   STATUS[439].EXT.AlarmSuppressed := FALSE;
   STATUS[439].EXT.AlarmPresent := FALSE;
   STATUS[439].EXT.AlarmFailUnAck := FALSE;
   STATUS[439].Status := 0;
   STATUS[439].TimeStamp := 16#0000;
   STATUS[440].EXT.AlarmWarnUnAck := FALSE;
   STATUS[440].EXT.AckRequired := FALSE;
   STATUS[440].EXT.Maintanence := FALSE;
   STATUS[440].EXT.Operation := FALSE;
   STATUS[440].EXT.Forced := FALSE;
   STATUS[440].EXT.BIT29 := FALSE;
   STATUS[440].EXT.BIT30 := FALSE;
   STATUS[440].EXT.BIT31 := FALSE;
   STATUS[440].EXT.ModeBit1 := FALSE;
   STATUS[440].EXT.ModeBit2 := FALSE;
   STATUS[440].EXT.ModeBit3 := FALSE;
   STATUS[440].EXT.BIT19 := FALSE;
   STATUS[440].EXT.BIT20 := FALSE;
   STATUS[440].EXT.AlarmSuppressed := FALSE;
   STATUS[440].EXT.AlarmPresent := FALSE;
   STATUS[440].EXT.AlarmFailUnAck := FALSE;
   STATUS[440].Status := 0;
   STATUS[440].TimeStamp := 16#0000;
   STATUS[441].EXT.AlarmWarnUnAck := FALSE;
   STATUS[441].EXT.AckRequired := FALSE;
   STATUS[441].EXT.Maintanence := FALSE;
   STATUS[441].EXT.Operation := FALSE;
   STATUS[441].EXT.Forced := FALSE;
   STATUS[441].EXT.BIT29 := FALSE;
   STATUS[441].EXT.BIT30 := FALSE;
   STATUS[441].EXT.BIT31 := FALSE;
   STATUS[441].EXT.ModeBit1 := FALSE;
   STATUS[441].EXT.ModeBit2 := FALSE;
   STATUS[441].EXT.ModeBit3 := FALSE;
   STATUS[441].EXT.BIT19 := FALSE;
   STATUS[441].EXT.BIT20 := FALSE;
   STATUS[441].EXT.AlarmSuppressed := FALSE;
   STATUS[441].EXT.AlarmPresent := FALSE;
   STATUS[441].EXT.AlarmFailUnAck := FALSE;
   STATUS[441].Status := 0;
   STATUS[441].TimeStamp := 16#0000;
   STATUS[442].EXT.AlarmWarnUnAck := FALSE;
   STATUS[442].EXT.AckRequired := FALSE;
   STATUS[442].EXT.Maintanence := FALSE;
   STATUS[442].EXT.Operation := FALSE;
   STATUS[442].EXT.Forced := FALSE;
   STATUS[442].EXT.BIT29 := FALSE;
   STATUS[442].EXT.BIT30 := FALSE;
   STATUS[442].EXT.BIT31 := FALSE;
   STATUS[442].EXT.ModeBit1 := FALSE;
   STATUS[442].EXT.ModeBit2 := FALSE;
   STATUS[442].EXT.ModeBit3 := FALSE;
   STATUS[442].EXT.BIT19 := FALSE;
   STATUS[442].EXT.BIT20 := FALSE;
   STATUS[442].EXT.AlarmSuppressed := FALSE;
   STATUS[442].EXT.AlarmPresent := FALSE;
   STATUS[442].EXT.AlarmFailUnAck := FALSE;
   STATUS[442].Status := 0;
   STATUS[442].TimeStamp := 16#0000;
   STATUS[443].EXT.AlarmWarnUnAck := FALSE;
   STATUS[443].EXT.AckRequired := FALSE;
   STATUS[443].EXT.Maintanence := FALSE;
   STATUS[443].EXT.Operation := FALSE;
   STATUS[443].EXT.Forced := FALSE;
   STATUS[443].EXT.BIT29 := FALSE;
   STATUS[443].EXT.BIT30 := FALSE;
   STATUS[443].EXT.BIT31 := FALSE;
   STATUS[443].EXT.ModeBit1 := FALSE;
   STATUS[443].EXT.ModeBit2 := FALSE;
   STATUS[443].EXT.ModeBit3 := FALSE;
   STATUS[443].EXT.BIT19 := FALSE;
   STATUS[443].EXT.BIT20 := FALSE;
   STATUS[443].EXT.AlarmSuppressed := FALSE;
   STATUS[443].EXT.AlarmPresent := FALSE;
   STATUS[443].EXT.AlarmFailUnAck := FALSE;
   STATUS[443].Status := 0;
   STATUS[443].TimeStamp := 16#0000;
   STATUS[444].EXT.AlarmWarnUnAck := FALSE;
   STATUS[444].EXT.AckRequired := FALSE;
   STATUS[444].EXT.Maintanence := FALSE;
   STATUS[444].EXT.Operation := FALSE;
   STATUS[444].EXT.Forced := FALSE;
   STATUS[444].EXT.BIT29 := FALSE;
   STATUS[444].EXT.BIT30 := FALSE;
   STATUS[444].EXT.BIT31 := FALSE;
   STATUS[444].EXT.ModeBit1 := FALSE;
   STATUS[444].EXT.ModeBit2 := FALSE;
   STATUS[444].EXT.ModeBit3 := FALSE;
   STATUS[444].EXT.BIT19 := FALSE;
   STATUS[444].EXT.BIT20 := FALSE;
   STATUS[444].EXT.AlarmSuppressed := FALSE;
   STATUS[444].EXT.AlarmPresent := FALSE;
   STATUS[444].EXT.AlarmFailUnAck := FALSE;
   STATUS[444].Status := 0;
   STATUS[444].TimeStamp := 16#0000;
   STATUS[445].EXT.AlarmWarnUnAck := FALSE;
   STATUS[445].EXT.AckRequired := FALSE;
   STATUS[445].EXT.Maintanence := FALSE;
   STATUS[445].EXT.Operation := FALSE;
   STATUS[445].EXT.Forced := FALSE;
   STATUS[445].EXT.BIT29 := FALSE;
   STATUS[445].EXT.BIT30 := FALSE;
   STATUS[445].EXT.BIT31 := FALSE;
   STATUS[445].EXT.ModeBit1 := FALSE;
   STATUS[445].EXT.ModeBit2 := FALSE;
   STATUS[445].EXT.ModeBit3 := FALSE;
   STATUS[445].EXT.BIT19 := FALSE;
   STATUS[445].EXT.BIT20 := FALSE;
   STATUS[445].EXT.AlarmSuppressed := FALSE;
   STATUS[445].EXT.AlarmPresent := FALSE;
   STATUS[445].EXT.AlarmFailUnAck := FALSE;
   STATUS[445].Status := 0;
   STATUS[445].TimeStamp := 16#0000;
   STATUS[446].EXT.AlarmWarnUnAck := FALSE;
   STATUS[446].EXT.AckRequired := FALSE;
   STATUS[446].EXT.Maintanence := FALSE;
   STATUS[446].EXT.Operation := FALSE;
   STATUS[446].EXT.Forced := FALSE;
   STATUS[446].EXT.BIT29 := FALSE;
   STATUS[446].EXT.BIT30 := FALSE;
   STATUS[446].EXT.BIT31 := FALSE;
   STATUS[446].EXT.ModeBit1 := FALSE;
   STATUS[446].EXT.ModeBit2 := FALSE;
   STATUS[446].EXT.ModeBit3 := FALSE;
   STATUS[446].EXT.BIT19 := FALSE;
   STATUS[446].EXT.BIT20 := FALSE;
   STATUS[446].EXT.AlarmSuppressed := FALSE;
   STATUS[446].EXT.AlarmPresent := FALSE;
   STATUS[446].EXT.AlarmFailUnAck := FALSE;
   STATUS[446].Status := 0;
   STATUS[446].TimeStamp := 16#0000;
   STATUS[447].EXT.AlarmWarnUnAck := FALSE;
   STATUS[447].EXT.AckRequired := FALSE;
   STATUS[447].EXT.Maintanence := FALSE;
   STATUS[447].EXT.Operation := FALSE;
   STATUS[447].EXT.Forced := FALSE;
   STATUS[447].EXT.BIT29 := FALSE;
   STATUS[447].EXT.BIT30 := FALSE;
   STATUS[447].EXT.BIT31 := FALSE;
   STATUS[447].EXT.ModeBit1 := FALSE;
   STATUS[447].EXT.ModeBit2 := FALSE;
   STATUS[447].EXT.ModeBit3 := FALSE;
   STATUS[447].EXT.BIT19 := FALSE;
   STATUS[447].EXT.BIT20 := FALSE;
   STATUS[447].EXT.AlarmSuppressed := FALSE;
   STATUS[447].EXT.AlarmPresent := FALSE;
   STATUS[447].EXT.AlarmFailUnAck := FALSE;
   STATUS[447].Status := 0;
   STATUS[447].TimeStamp := 16#0000;
   STATUS[448].EXT.AlarmWarnUnAck := FALSE;
   STATUS[448].EXT.AckRequired := FALSE;
   STATUS[448].EXT.Maintanence := FALSE;
   STATUS[448].EXT.Operation := FALSE;
   STATUS[448].EXT.Forced := FALSE;
   STATUS[448].EXT.BIT29 := FALSE;
   STATUS[448].EXT.BIT30 := FALSE;
   STATUS[448].EXT.BIT31 := FALSE;
   STATUS[448].EXT.ModeBit1 := FALSE;
   STATUS[448].EXT.ModeBit2 := FALSE;
   STATUS[448].EXT.ModeBit3 := FALSE;
   STATUS[448].EXT.BIT19 := FALSE;
   STATUS[448].EXT.BIT20 := FALSE;
   STATUS[448].EXT.AlarmSuppressed := FALSE;
   STATUS[448].EXT.AlarmPresent := FALSE;
   STATUS[448].EXT.AlarmFailUnAck := FALSE;
   STATUS[448].Status := 0;
   STATUS[448].TimeStamp := 16#0000;
   STATUS[449].EXT.AlarmWarnUnAck := FALSE;
   STATUS[449].EXT.AckRequired := FALSE;
   STATUS[449].EXT.Maintanence := FALSE;
   STATUS[449].EXT.Operation := FALSE;
   STATUS[449].EXT.Forced := FALSE;
   STATUS[449].EXT.BIT29 := FALSE;
   STATUS[449].EXT.BIT30 := FALSE;
   STATUS[449].EXT.BIT31 := FALSE;
   STATUS[449].EXT.ModeBit1 := FALSE;
   STATUS[449].EXT.ModeBit2 := FALSE;
   STATUS[449].EXT.ModeBit3 := FALSE;
   STATUS[449].EXT.BIT19 := FALSE;
   STATUS[449].EXT.BIT20 := FALSE;
   STATUS[449].EXT.AlarmSuppressed := FALSE;
   STATUS[449].EXT.AlarmPresent := FALSE;
   STATUS[449].EXT.AlarmFailUnAck := FALSE;
   STATUS[449].Status := 0;
   STATUS[449].TimeStamp := 16#0000;
   STATUS[450].EXT.AlarmWarnUnAck := FALSE;
   STATUS[450].EXT.AckRequired := FALSE;
   STATUS[450].EXT.Maintanence := FALSE;
   STATUS[450].EXT.Operation := FALSE;
   STATUS[450].EXT.Forced := FALSE;
   STATUS[450].EXT.BIT29 := FALSE;
   STATUS[450].EXT.BIT30 := FALSE;
   STATUS[450].EXT.BIT31 := FALSE;
   STATUS[450].EXT.ModeBit1 := FALSE;
   STATUS[450].EXT.ModeBit2 := FALSE;
   STATUS[450].EXT.ModeBit3 := FALSE;
   STATUS[450].EXT.BIT19 := FALSE;
   STATUS[450].EXT.BIT20 := FALSE;
   STATUS[450].EXT.AlarmSuppressed := FALSE;
   STATUS[450].EXT.AlarmPresent := FALSE;
   STATUS[450].EXT.AlarmFailUnAck := FALSE;
   STATUS[450].Status := 0;
   STATUS[450].TimeStamp := 16#0000;
   STATUS[451].EXT.AlarmWarnUnAck := FALSE;
   STATUS[451].EXT.AckRequired := FALSE;
   STATUS[451].EXT.Maintanence := FALSE;
   STATUS[451].EXT.Operation := FALSE;
   STATUS[451].EXT.Forced := FALSE;
   STATUS[451].EXT.BIT29 := FALSE;
   STATUS[451].EXT.BIT30 := FALSE;
   STATUS[451].EXT.BIT31 := FALSE;
   STATUS[451].EXT.ModeBit1 := FALSE;
   STATUS[451].EXT.ModeBit2 := FALSE;
   STATUS[451].EXT.ModeBit3 := FALSE;
   STATUS[451].EXT.BIT19 := FALSE;
   STATUS[451].EXT.BIT20 := FALSE;
   STATUS[451].EXT.AlarmSuppressed := FALSE;
   STATUS[451].EXT.AlarmPresent := FALSE;
   STATUS[451].EXT.AlarmFailUnAck := FALSE;
   STATUS[451].Status := 0;
   STATUS[451].TimeStamp := 16#0000;
   STATUS[452].EXT.AlarmWarnUnAck := FALSE;
   STATUS[452].EXT.AckRequired := FALSE;
   STATUS[452].EXT.Maintanence := FALSE;
   STATUS[452].EXT.Operation := FALSE;
   STATUS[452].EXT.Forced := FALSE;
   STATUS[452].EXT.BIT29 := FALSE;
   STATUS[452].EXT.BIT30 := FALSE;
   STATUS[452].EXT.BIT31 := FALSE;
   STATUS[452].EXT.ModeBit1 := FALSE;
   STATUS[452].EXT.ModeBit2 := FALSE;
   STATUS[452].EXT.ModeBit3 := FALSE;
   STATUS[452].EXT.BIT19 := FALSE;
   STATUS[452].EXT.BIT20 := FALSE;
   STATUS[452].EXT.AlarmSuppressed := FALSE;
   STATUS[452].EXT.AlarmPresent := FALSE;
   STATUS[452].EXT.AlarmFailUnAck := FALSE;
   STATUS[452].Status := 0;
   STATUS[452].TimeStamp := 16#0000;
   STATUS[453].EXT.AlarmWarnUnAck := FALSE;
   STATUS[453].EXT.AckRequired := FALSE;
   STATUS[453].EXT.Maintanence := FALSE;
   STATUS[453].EXT.Operation := FALSE;
   STATUS[453].EXT.Forced := FALSE;
   STATUS[453].EXT.BIT29 := FALSE;
   STATUS[453].EXT.BIT30 := FALSE;
   STATUS[453].EXT.BIT31 := FALSE;
   STATUS[453].EXT.ModeBit1 := FALSE;
   STATUS[453].EXT.ModeBit2 := FALSE;
   STATUS[453].EXT.ModeBit3 := FALSE;
   STATUS[453].EXT.BIT19 := FALSE;
   STATUS[453].EXT.BIT20 := FALSE;
   STATUS[453].EXT.AlarmSuppressed := FALSE;
   STATUS[453].EXT.AlarmPresent := FALSE;
   STATUS[453].EXT.AlarmFailUnAck := FALSE;
   STATUS[453].Status := 0;
   STATUS[453].TimeStamp := 16#0000;
   STATUS[454].EXT.AlarmWarnUnAck := FALSE;
   STATUS[454].EXT.AckRequired := FALSE;
   STATUS[454].EXT.Maintanence := FALSE;
   STATUS[454].EXT.Operation := FALSE;
   STATUS[454].EXT.Forced := FALSE;
   STATUS[454].EXT.BIT29 := FALSE;
   STATUS[454].EXT.BIT30 := FALSE;
   STATUS[454].EXT.BIT31 := FALSE;
   STATUS[454].EXT.ModeBit1 := FALSE;
   STATUS[454].EXT.ModeBit2 := FALSE;
   STATUS[454].EXT.ModeBit3 := FALSE;
   STATUS[454].EXT.BIT19 := FALSE;
   STATUS[454].EXT.BIT20 := FALSE;
   STATUS[454].EXT.AlarmSuppressed := FALSE;
   STATUS[454].EXT.AlarmPresent := FALSE;
   STATUS[454].EXT.AlarmFailUnAck := FALSE;
   STATUS[454].Status := 0;
   STATUS[454].TimeStamp := 16#0000;
   STATUS[455].EXT.AlarmWarnUnAck := FALSE;
   STATUS[455].EXT.AckRequired := FALSE;
   STATUS[455].EXT.Maintanence := FALSE;
   STATUS[455].EXT.Operation := FALSE;
   STATUS[455].EXT.Forced := FALSE;
   STATUS[455].EXT.BIT29 := FALSE;
   STATUS[455].EXT.BIT30 := FALSE;
   STATUS[455].EXT.BIT31 := FALSE;
   STATUS[455].EXT.ModeBit1 := FALSE;
   STATUS[455].EXT.ModeBit2 := FALSE;
   STATUS[455].EXT.ModeBit3 := FALSE;
   STATUS[455].EXT.BIT19 := FALSE;
   STATUS[455].EXT.BIT20 := FALSE;
   STATUS[455].EXT.AlarmSuppressed := FALSE;
   STATUS[455].EXT.AlarmPresent := FALSE;
   STATUS[455].EXT.AlarmFailUnAck := FALSE;
   STATUS[455].Status := 0;
   STATUS[455].TimeStamp := 16#0000;
   STATUS[456].EXT.AlarmWarnUnAck := FALSE;
   STATUS[456].EXT.AckRequired := FALSE;
   STATUS[456].EXT.Maintanence := FALSE;
   STATUS[456].EXT.Operation := FALSE;
   STATUS[456].EXT.Forced := FALSE;
   STATUS[456].EXT.BIT29 := FALSE;
   STATUS[456].EXT.BIT30 := FALSE;
   STATUS[456].EXT.BIT31 := FALSE;
   STATUS[456].EXT.ModeBit1 := FALSE;
   STATUS[456].EXT.ModeBit2 := FALSE;
   STATUS[456].EXT.ModeBit3 := FALSE;
   STATUS[456].EXT.BIT19 := FALSE;
   STATUS[456].EXT.BIT20 := FALSE;
   STATUS[456].EXT.AlarmSuppressed := FALSE;
   STATUS[456].EXT.AlarmPresent := FALSE;
   STATUS[456].EXT.AlarmFailUnAck := FALSE;
   STATUS[456].Status := 0;
   STATUS[456].TimeStamp := 16#0000;
   STATUS[457].EXT.AlarmWarnUnAck := FALSE;
   STATUS[457].EXT.AckRequired := FALSE;
   STATUS[457].EXT.Maintanence := FALSE;
   STATUS[457].EXT.Operation := FALSE;
   STATUS[457].EXT.Forced := FALSE;
   STATUS[457].EXT.BIT29 := FALSE;
   STATUS[457].EXT.BIT30 := FALSE;
   STATUS[457].EXT.BIT31 := FALSE;
   STATUS[457].EXT.ModeBit1 := FALSE;
   STATUS[457].EXT.ModeBit2 := FALSE;
   STATUS[457].EXT.ModeBit3 := FALSE;
   STATUS[457].EXT.BIT19 := FALSE;
   STATUS[457].EXT.BIT20 := FALSE;
   STATUS[457].EXT.AlarmSuppressed := FALSE;
   STATUS[457].EXT.AlarmPresent := FALSE;
   STATUS[457].EXT.AlarmFailUnAck := FALSE;
   STATUS[457].Status := 0;
   STATUS[457].TimeStamp := 16#0000;
   STATUS[458].EXT.AlarmWarnUnAck := FALSE;
   STATUS[458].EXT.AckRequired := FALSE;
   STATUS[458].EXT.Maintanence := FALSE;
   STATUS[458].EXT.Operation := FALSE;
   STATUS[458].EXT.Forced := FALSE;
   STATUS[458].EXT.BIT29 := FALSE;
   STATUS[458].EXT.BIT30 := FALSE;
   STATUS[458].EXT.BIT31 := FALSE;
   STATUS[458].EXT.ModeBit1 := FALSE;
   STATUS[458].EXT.ModeBit2 := FALSE;
   STATUS[458].EXT.ModeBit3 := FALSE;
   STATUS[458].EXT.BIT19 := FALSE;
   STATUS[458].EXT.BIT20 := FALSE;
   STATUS[458].EXT.AlarmSuppressed := FALSE;
   STATUS[458].EXT.AlarmPresent := FALSE;
   STATUS[458].EXT.AlarmFailUnAck := FALSE;
   STATUS[458].Status := 0;
   STATUS[458].TimeStamp := 16#0000;
   STATUS[459].EXT.AlarmWarnUnAck := FALSE;
   STATUS[459].EXT.AckRequired := FALSE;
   STATUS[459].EXT.Maintanence := FALSE;
   STATUS[459].EXT.Operation := FALSE;
   STATUS[459].EXT.Forced := FALSE;
   STATUS[459].EXT.BIT29 := FALSE;
   STATUS[459].EXT.BIT30 := FALSE;
   STATUS[459].EXT.BIT31 := FALSE;
   STATUS[459].EXT.ModeBit1 := FALSE;
   STATUS[459].EXT.ModeBit2 := FALSE;
   STATUS[459].EXT.ModeBit3 := FALSE;
   STATUS[459].EXT.BIT19 := FALSE;
   STATUS[459].EXT.BIT20 := FALSE;
   STATUS[459].EXT.AlarmSuppressed := FALSE;
   STATUS[459].EXT.AlarmPresent := FALSE;
   STATUS[459].EXT.AlarmFailUnAck := FALSE;
   STATUS[459].Status := 0;
   STATUS[459].TimeStamp := 16#0000;
   STATUS[460].EXT.AlarmWarnUnAck := FALSE;
   STATUS[460].EXT.AckRequired := FALSE;
   STATUS[460].EXT.Maintanence := FALSE;
   STATUS[460].EXT.Operation := FALSE;
   STATUS[460].EXT.Forced := FALSE;
   STATUS[460].EXT.BIT29 := FALSE;
   STATUS[460].EXT.BIT30 := FALSE;
   STATUS[460].EXT.BIT31 := FALSE;
   STATUS[460].EXT.ModeBit1 := FALSE;
   STATUS[460].EXT.ModeBit2 := FALSE;
   STATUS[460].EXT.ModeBit3 := FALSE;
   STATUS[460].EXT.BIT19 := FALSE;
   STATUS[460].EXT.BIT20 := FALSE;
   STATUS[460].EXT.AlarmSuppressed := FALSE;
   STATUS[460].EXT.AlarmPresent := FALSE;
   STATUS[460].EXT.AlarmFailUnAck := FALSE;
   STATUS[460].Status := 0;
   STATUS[460].TimeStamp := 16#0000;
   STATUS[461].EXT.AlarmWarnUnAck := FALSE;
   STATUS[461].EXT.AckRequired := FALSE;
   STATUS[461].EXT.Maintanence := FALSE;
   STATUS[461].EXT.Operation := FALSE;
   STATUS[461].EXT.Forced := FALSE;
   STATUS[461].EXT.BIT29 := FALSE;
   STATUS[461].EXT.BIT30 := FALSE;
   STATUS[461].EXT.BIT31 := FALSE;
   STATUS[461].EXT.ModeBit1 := FALSE;
   STATUS[461].EXT.ModeBit2 := FALSE;
   STATUS[461].EXT.ModeBit3 := FALSE;
   STATUS[461].EXT.BIT19 := FALSE;
   STATUS[461].EXT.BIT20 := FALSE;
   STATUS[461].EXT.AlarmSuppressed := FALSE;
   STATUS[461].EXT.AlarmPresent := FALSE;
   STATUS[461].EXT.AlarmFailUnAck := FALSE;
   STATUS[461].Status := 0;
   STATUS[461].TimeStamp := 16#0000;
   STATUS[462].EXT.AlarmWarnUnAck := FALSE;
   STATUS[462].EXT.AckRequired := FALSE;
   STATUS[462].EXT.Maintanence := FALSE;
   STATUS[462].EXT.Operation := FALSE;
   STATUS[462].EXT.Forced := FALSE;
   STATUS[462].EXT.BIT29 := FALSE;
   STATUS[462].EXT.BIT30 := FALSE;
   STATUS[462].EXT.BIT31 := FALSE;
   STATUS[462].EXT.ModeBit1 := FALSE;
   STATUS[462].EXT.ModeBit2 := FALSE;
   STATUS[462].EXT.ModeBit3 := FALSE;
   STATUS[462].EXT.BIT19 := FALSE;
   STATUS[462].EXT.BIT20 := FALSE;
   STATUS[462].EXT.AlarmSuppressed := FALSE;
   STATUS[462].EXT.AlarmPresent := FALSE;
   STATUS[462].EXT.AlarmFailUnAck := FALSE;
   STATUS[462].Status := 0;
   STATUS[462].TimeStamp := 16#0000;
   STATUS[463].EXT.AlarmWarnUnAck := FALSE;
   STATUS[463].EXT.AckRequired := FALSE;
   STATUS[463].EXT.Maintanence := FALSE;
   STATUS[463].EXT.Operation := FALSE;
   STATUS[463].EXT.Forced := FALSE;
   STATUS[463].EXT.BIT29 := FALSE;
   STATUS[463].EXT.BIT30 := FALSE;
   STATUS[463].EXT.BIT31 := FALSE;
   STATUS[463].EXT.ModeBit1 := FALSE;
   STATUS[463].EXT.ModeBit2 := FALSE;
   STATUS[463].EXT.ModeBit3 := FALSE;
   STATUS[463].EXT.BIT19 := FALSE;
   STATUS[463].EXT.BIT20 := FALSE;
   STATUS[463].EXT.AlarmSuppressed := FALSE;
   STATUS[463].EXT.AlarmPresent := FALSE;
   STATUS[463].EXT.AlarmFailUnAck := FALSE;
   STATUS[463].Status := 0;
   STATUS[463].TimeStamp := 16#0000;
   STATUS[464].EXT.AlarmWarnUnAck := FALSE;
   STATUS[464].EXT.AckRequired := FALSE;
   STATUS[464].EXT.Maintanence := FALSE;
   STATUS[464].EXT.Operation := FALSE;
   STATUS[464].EXT.Forced := FALSE;
   STATUS[464].EXT.BIT29 := FALSE;
   STATUS[464].EXT.BIT30 := FALSE;
   STATUS[464].EXT.BIT31 := FALSE;
   STATUS[464].EXT.ModeBit1 := FALSE;
   STATUS[464].EXT.ModeBit2 := FALSE;
   STATUS[464].EXT.ModeBit3 := FALSE;
   STATUS[464].EXT.BIT19 := FALSE;
   STATUS[464].EXT.BIT20 := FALSE;
   STATUS[464].EXT.AlarmSuppressed := FALSE;
   STATUS[464].EXT.AlarmPresent := FALSE;
   STATUS[464].EXT.AlarmFailUnAck := FALSE;
   STATUS[464].Status := 0;
   STATUS[464].TimeStamp := 16#0000;
   STATUS[465].EXT.AlarmWarnUnAck := FALSE;
   STATUS[465].EXT.AckRequired := FALSE;
   STATUS[465].EXT.Maintanence := FALSE;
   STATUS[465].EXT.Operation := FALSE;
   STATUS[465].EXT.Forced := FALSE;
   STATUS[465].EXT.BIT29 := FALSE;
   STATUS[465].EXT.BIT30 := FALSE;
   STATUS[465].EXT.BIT31 := FALSE;
   STATUS[465].EXT.ModeBit1 := FALSE;
   STATUS[465].EXT.ModeBit2 := FALSE;
   STATUS[465].EXT.ModeBit3 := FALSE;
   STATUS[465].EXT.BIT19 := FALSE;
   STATUS[465].EXT.BIT20 := FALSE;
   STATUS[465].EXT.AlarmSuppressed := FALSE;
   STATUS[465].EXT.AlarmPresent := FALSE;
   STATUS[465].EXT.AlarmFailUnAck := FALSE;
   STATUS[465].Status := 0;
   STATUS[465].TimeStamp := 16#0000;
   STATUS[466].EXT.AlarmWarnUnAck := FALSE;
   STATUS[466].EXT.AckRequired := FALSE;
   STATUS[466].EXT.Maintanence := FALSE;
   STATUS[466].EXT.Operation := FALSE;
   STATUS[466].EXT.Forced := FALSE;
   STATUS[466].EXT.BIT29 := FALSE;
   STATUS[466].EXT.BIT30 := FALSE;
   STATUS[466].EXT.BIT31 := FALSE;
   STATUS[466].EXT.ModeBit1 := FALSE;
   STATUS[466].EXT.ModeBit2 := FALSE;
   STATUS[466].EXT.ModeBit3 := FALSE;
   STATUS[466].EXT.BIT19 := FALSE;
   STATUS[466].EXT.BIT20 := FALSE;
   STATUS[466].EXT.AlarmSuppressed := FALSE;
   STATUS[466].EXT.AlarmPresent := FALSE;
   STATUS[466].EXT.AlarmFailUnAck := FALSE;
   STATUS[466].Status := 0;
   STATUS[466].TimeStamp := 16#0000;
   STATUS[467].EXT.AlarmWarnUnAck := FALSE;
   STATUS[467].EXT.AckRequired := FALSE;
   STATUS[467].EXT.Maintanence := FALSE;
   STATUS[467].EXT.Operation := FALSE;
   STATUS[467].EXT.Forced := FALSE;
   STATUS[467].EXT.BIT29 := FALSE;
   STATUS[467].EXT.BIT30 := FALSE;
   STATUS[467].EXT.BIT31 := FALSE;
   STATUS[467].EXT.ModeBit1 := FALSE;
   STATUS[467].EXT.ModeBit2 := FALSE;
   STATUS[467].EXT.ModeBit3 := FALSE;
   STATUS[467].EXT.BIT19 := FALSE;
   STATUS[467].EXT.BIT20 := FALSE;
   STATUS[467].EXT.AlarmSuppressed := FALSE;
   STATUS[467].EXT.AlarmPresent := FALSE;
   STATUS[467].EXT.AlarmFailUnAck := FALSE;
   STATUS[467].Status := 0;
   STATUS[467].TimeStamp := 16#0000;
   STATUS[468].EXT.AlarmWarnUnAck := FALSE;
   STATUS[468].EXT.AckRequired := FALSE;
   STATUS[468].EXT.Maintanence := FALSE;
   STATUS[468].EXT.Operation := FALSE;
   STATUS[468].EXT.Forced := FALSE;
   STATUS[468].EXT.BIT29 := FALSE;
   STATUS[468].EXT.BIT30 := FALSE;
   STATUS[468].EXT.BIT31 := FALSE;
   STATUS[468].EXT.ModeBit1 := FALSE;
   STATUS[468].EXT.ModeBit2 := FALSE;
   STATUS[468].EXT.ModeBit3 := FALSE;
   STATUS[468].EXT.BIT19 := FALSE;
   STATUS[468].EXT.BIT20 := FALSE;
   STATUS[468].EXT.AlarmSuppressed := FALSE;
   STATUS[468].EXT.AlarmPresent := FALSE;
   STATUS[468].EXT.AlarmFailUnAck := FALSE;
   STATUS[468].Status := 0;
   STATUS[468].TimeStamp := 16#0000;
   STATUS[469].EXT.AlarmWarnUnAck := FALSE;
   STATUS[469].EXT.AckRequired := FALSE;
   STATUS[469].EXT.Maintanence := FALSE;
   STATUS[469].EXT.Operation := FALSE;
   STATUS[469].EXT.Forced := FALSE;
   STATUS[469].EXT.BIT29 := FALSE;
   STATUS[469].EXT.BIT30 := FALSE;
   STATUS[469].EXT.BIT31 := FALSE;
   STATUS[469].EXT.ModeBit1 := FALSE;
   STATUS[469].EXT.ModeBit2 := FALSE;
   STATUS[469].EXT.ModeBit3 := FALSE;
   STATUS[469].EXT.BIT19 := FALSE;
   STATUS[469].EXT.BIT20 := FALSE;
   STATUS[469].EXT.AlarmSuppressed := FALSE;
   STATUS[469].EXT.AlarmPresent := FALSE;
   STATUS[469].EXT.AlarmFailUnAck := FALSE;
   STATUS[469].Status := 0;
   STATUS[469].TimeStamp := 16#0000;
   STATUS[470].EXT.AlarmWarnUnAck := FALSE;
   STATUS[470].EXT.AckRequired := FALSE;
   STATUS[470].EXT.Maintanence := FALSE;
   STATUS[470].EXT.Operation := FALSE;
   STATUS[470].EXT.Forced := FALSE;
   STATUS[470].EXT.BIT29 := FALSE;
   STATUS[470].EXT.BIT30 := FALSE;
   STATUS[470].EXT.BIT31 := FALSE;
   STATUS[470].EXT.ModeBit1 := FALSE;
   STATUS[470].EXT.ModeBit2 := FALSE;
   STATUS[470].EXT.ModeBit3 := FALSE;
   STATUS[470].EXT.BIT19 := FALSE;
   STATUS[470].EXT.BIT20 := FALSE;
   STATUS[470].EXT.AlarmSuppressed := FALSE;
   STATUS[470].EXT.AlarmPresent := FALSE;
   STATUS[470].EXT.AlarmFailUnAck := FALSE;
   STATUS[470].Status := 0;
   STATUS[470].TimeStamp := 16#0000;
   STATUS[471].EXT.AlarmWarnUnAck := FALSE;
   STATUS[471].EXT.AckRequired := FALSE;
   STATUS[471].EXT.Maintanence := FALSE;
   STATUS[471].EXT.Operation := FALSE;
   STATUS[471].EXT.Forced := FALSE;
   STATUS[471].EXT.BIT29 := FALSE;
   STATUS[471].EXT.BIT30 := FALSE;
   STATUS[471].EXT.BIT31 := FALSE;
   STATUS[471].EXT.ModeBit1 := FALSE;
   STATUS[471].EXT.ModeBit2 := FALSE;
   STATUS[471].EXT.ModeBit3 := FALSE;
   STATUS[471].EXT.BIT19 := FALSE;
   STATUS[471].EXT.BIT20 := FALSE;
   STATUS[471].EXT.AlarmSuppressed := FALSE;
   STATUS[471].EXT.AlarmPresent := FALSE;
   STATUS[471].EXT.AlarmFailUnAck := FALSE;
   STATUS[471].Status := 0;
   STATUS[471].TimeStamp := 16#0000;
   STATUS[472].EXT.AlarmWarnUnAck := FALSE;
   STATUS[472].EXT.AckRequired := FALSE;
   STATUS[472].EXT.Maintanence := FALSE;
   STATUS[472].EXT.Operation := FALSE;
   STATUS[472].EXT.Forced := FALSE;
   STATUS[472].EXT.BIT29 := FALSE;
   STATUS[472].EXT.BIT30 := FALSE;
   STATUS[472].EXT.BIT31 := FALSE;
   STATUS[472].EXT.ModeBit1 := FALSE;
   STATUS[472].EXT.ModeBit2 := FALSE;
   STATUS[472].EXT.ModeBit3 := FALSE;
   STATUS[472].EXT.BIT19 := FALSE;
   STATUS[472].EXT.BIT20 := FALSE;
   STATUS[472].EXT.AlarmSuppressed := FALSE;
   STATUS[472].EXT.AlarmPresent := FALSE;
   STATUS[472].EXT.AlarmFailUnAck := FALSE;
   STATUS[472].Status := 0;
   STATUS[472].TimeStamp := 16#0000;
   STATUS[473].EXT.AlarmWarnUnAck := FALSE;
   STATUS[473].EXT.AckRequired := FALSE;
   STATUS[473].EXT.Maintanence := FALSE;
   STATUS[473].EXT.Operation := FALSE;
   STATUS[473].EXT.Forced := FALSE;
   STATUS[473].EXT.BIT29 := FALSE;
   STATUS[473].EXT.BIT30 := FALSE;
   STATUS[473].EXT.BIT31 := FALSE;
   STATUS[473].EXT.ModeBit1 := FALSE;
   STATUS[473].EXT.ModeBit2 := FALSE;
   STATUS[473].EXT.ModeBit3 := FALSE;
   STATUS[473].EXT.BIT19 := FALSE;
   STATUS[473].EXT.BIT20 := FALSE;
   STATUS[473].EXT.AlarmSuppressed := FALSE;
   STATUS[473].EXT.AlarmPresent := FALSE;
   STATUS[473].EXT.AlarmFailUnAck := FALSE;
   STATUS[473].Status := 0;
   STATUS[473].TimeStamp := 16#0000;
   STATUS[474].EXT.AlarmWarnUnAck := FALSE;
   STATUS[474].EXT.AckRequired := FALSE;
   STATUS[474].EXT.Maintanence := FALSE;
   STATUS[474].EXT.Operation := FALSE;
   STATUS[474].EXT.Forced := FALSE;
   STATUS[474].EXT.BIT29 := FALSE;
   STATUS[474].EXT.BIT30 := FALSE;
   STATUS[474].EXT.BIT31 := FALSE;
   STATUS[474].EXT.ModeBit1 := FALSE;
   STATUS[474].EXT.ModeBit2 := FALSE;
   STATUS[474].EXT.ModeBit3 := FALSE;
   STATUS[474].EXT.BIT19 := FALSE;
   STATUS[474].EXT.BIT20 := FALSE;
   STATUS[474].EXT.AlarmSuppressed := FALSE;
   STATUS[474].EXT.AlarmPresent := FALSE;
   STATUS[474].EXT.AlarmFailUnAck := FALSE;
   STATUS[474].Status := 0;
   STATUS[474].TimeStamp := 16#0000;
   STATUS[475].EXT.AlarmWarnUnAck := FALSE;
   STATUS[475].EXT.AckRequired := FALSE;
   STATUS[475].EXT.Maintanence := FALSE;
   STATUS[475].EXT.Operation := FALSE;
   STATUS[475].EXT.Forced := FALSE;
   STATUS[475].EXT.BIT29 := FALSE;
   STATUS[475].EXT.BIT30 := FALSE;
   STATUS[475].EXT.BIT31 := FALSE;
   STATUS[475].EXT.ModeBit1 := FALSE;
   STATUS[475].EXT.ModeBit2 := FALSE;
   STATUS[475].EXT.ModeBit3 := FALSE;
   STATUS[475].EXT.BIT19 := FALSE;
   STATUS[475].EXT.BIT20 := FALSE;
   STATUS[475].EXT.AlarmSuppressed := FALSE;
   STATUS[475].EXT.AlarmPresent := FALSE;
   STATUS[475].EXT.AlarmFailUnAck := FALSE;
   STATUS[475].Status := 0;
   STATUS[475].TimeStamp := 16#0000;
   STATUS[476].EXT.AlarmWarnUnAck := FALSE;
   STATUS[476].EXT.AckRequired := FALSE;
   STATUS[476].EXT.Maintanence := FALSE;
   STATUS[476].EXT.Operation := FALSE;
   STATUS[476].EXT.Forced := FALSE;
   STATUS[476].EXT.BIT29 := FALSE;
   STATUS[476].EXT.BIT30 := FALSE;
   STATUS[476].EXT.BIT31 := FALSE;
   STATUS[476].EXT.ModeBit1 := FALSE;
   STATUS[476].EXT.ModeBit2 := FALSE;
   STATUS[476].EXT.ModeBit3 := FALSE;
   STATUS[476].EXT.BIT19 := FALSE;
   STATUS[476].EXT.BIT20 := FALSE;
   STATUS[476].EXT.AlarmSuppressed := FALSE;
   STATUS[476].EXT.AlarmPresent := FALSE;
   STATUS[476].EXT.AlarmFailUnAck := FALSE;
   STATUS[476].Status := 0;
   STATUS[476].TimeStamp := 16#0000;
   STATUS[477].EXT.AlarmWarnUnAck := FALSE;
   STATUS[477].EXT.AckRequired := FALSE;
   STATUS[477].EXT.Maintanence := FALSE;
   STATUS[477].EXT.Operation := FALSE;
   STATUS[477].EXT.Forced := FALSE;
   STATUS[477].EXT.BIT29 := FALSE;
   STATUS[477].EXT.BIT30 := FALSE;
   STATUS[477].EXT.BIT31 := FALSE;
   STATUS[477].EXT.ModeBit1 := FALSE;
   STATUS[477].EXT.ModeBit2 := FALSE;
   STATUS[477].EXT.ModeBit3 := FALSE;
   STATUS[477].EXT.BIT19 := FALSE;
   STATUS[477].EXT.BIT20 := FALSE;
   STATUS[477].EXT.AlarmSuppressed := FALSE;
   STATUS[477].EXT.AlarmPresent := FALSE;
   STATUS[477].EXT.AlarmFailUnAck := FALSE;
   STATUS[477].Status := 0;
   STATUS[477].TimeStamp := 16#0000;
   STATUS[478].EXT.AlarmWarnUnAck := FALSE;
   STATUS[478].EXT.AckRequired := FALSE;
   STATUS[478].EXT.Maintanence := FALSE;
   STATUS[478].EXT.Operation := FALSE;
   STATUS[478].EXT.Forced := FALSE;
   STATUS[478].EXT.BIT29 := FALSE;
   STATUS[478].EXT.BIT30 := FALSE;
   STATUS[478].EXT.BIT31 := FALSE;
   STATUS[478].EXT.ModeBit1 := FALSE;
   STATUS[478].EXT.ModeBit2 := FALSE;
   STATUS[478].EXT.ModeBit3 := FALSE;
   STATUS[478].EXT.BIT19 := FALSE;
   STATUS[478].EXT.BIT20 := FALSE;
   STATUS[478].EXT.AlarmSuppressed := FALSE;
   STATUS[478].EXT.AlarmPresent := FALSE;
   STATUS[478].EXT.AlarmFailUnAck := FALSE;
   STATUS[478].Status := 0;
   STATUS[478].TimeStamp := 16#0000;
   STATUS[479].EXT.AlarmWarnUnAck := FALSE;
   STATUS[479].EXT.AckRequired := FALSE;
   STATUS[479].EXT.Maintanence := FALSE;
   STATUS[479].EXT.Operation := FALSE;
   STATUS[479].EXT.Forced := FALSE;
   STATUS[479].EXT.BIT29 := FALSE;
   STATUS[479].EXT.BIT30 := FALSE;
   STATUS[479].EXT.BIT31 := FALSE;
   STATUS[479].EXT.ModeBit1 := FALSE;
   STATUS[479].EXT.ModeBit2 := FALSE;
   STATUS[479].EXT.ModeBit3 := FALSE;
   STATUS[479].EXT.BIT19 := FALSE;
   STATUS[479].EXT.BIT20 := FALSE;
   STATUS[479].EXT.AlarmSuppressed := FALSE;
   STATUS[479].EXT.AlarmPresent := FALSE;
   STATUS[479].EXT.AlarmFailUnAck := FALSE;
   STATUS[479].Status := 0;
   STATUS[479].TimeStamp := 16#0000;
   STATUS[480].EXT.AlarmWarnUnAck := FALSE;
   STATUS[480].EXT.AckRequired := FALSE;
   STATUS[480].EXT.Maintanence := FALSE;
   STATUS[480].EXT.Operation := FALSE;
   STATUS[480].EXT.Forced := FALSE;
   STATUS[480].EXT.BIT29 := FALSE;
   STATUS[480].EXT.BIT30 := FALSE;
   STATUS[480].EXT.BIT31 := FALSE;
   STATUS[480].EXT.ModeBit1 := FALSE;
   STATUS[480].EXT.ModeBit2 := FALSE;
   STATUS[480].EXT.ModeBit3 := FALSE;
   STATUS[480].EXT.BIT19 := FALSE;
   STATUS[480].EXT.BIT20 := FALSE;
   STATUS[480].EXT.AlarmSuppressed := FALSE;
   STATUS[480].EXT.AlarmPresent := FALSE;
   STATUS[480].EXT.AlarmFailUnAck := FALSE;
   STATUS[480].Status := 0;
   STATUS[480].TimeStamp := 16#0000;
   STATUS[481].EXT.AlarmWarnUnAck := FALSE;
   STATUS[481].EXT.AckRequired := FALSE;
   STATUS[481].EXT.Maintanence := FALSE;
   STATUS[481].EXT.Operation := FALSE;
   STATUS[481].EXT.Forced := FALSE;
   STATUS[481].EXT.BIT29 := FALSE;
   STATUS[481].EXT.BIT30 := FALSE;
   STATUS[481].EXT.BIT31 := FALSE;
   STATUS[481].EXT.ModeBit1 := FALSE;
   STATUS[481].EXT.ModeBit2 := FALSE;
   STATUS[481].EXT.ModeBit3 := FALSE;
   STATUS[481].EXT.BIT19 := FALSE;
   STATUS[481].EXT.BIT20 := FALSE;
   STATUS[481].EXT.AlarmSuppressed := FALSE;
   STATUS[481].EXT.AlarmPresent := FALSE;
   STATUS[481].EXT.AlarmFailUnAck := FALSE;
   STATUS[481].Status := 0;
   STATUS[481].TimeStamp := 16#0000;
   STATUS[482].EXT.AlarmWarnUnAck := FALSE;
   STATUS[482].EXT.AckRequired := FALSE;
   STATUS[482].EXT.Maintanence := FALSE;
   STATUS[482].EXT.Operation := FALSE;
   STATUS[482].EXT.Forced := FALSE;
   STATUS[482].EXT.BIT29 := FALSE;
   STATUS[482].EXT.BIT30 := FALSE;
   STATUS[482].EXT.BIT31 := FALSE;
   STATUS[482].EXT.ModeBit1 := FALSE;
   STATUS[482].EXT.ModeBit2 := FALSE;
   STATUS[482].EXT.ModeBit3 := FALSE;
   STATUS[482].EXT.BIT19 := FALSE;
   STATUS[482].EXT.BIT20 := FALSE;
   STATUS[482].EXT.AlarmSuppressed := FALSE;
   STATUS[482].EXT.AlarmPresent := FALSE;
   STATUS[482].EXT.AlarmFailUnAck := FALSE;
   STATUS[482].Status := 0;
   STATUS[482].TimeStamp := 16#0000;
   STATUS[483].EXT.AlarmWarnUnAck := FALSE;
   STATUS[483].EXT.AckRequired := FALSE;
   STATUS[483].EXT.Maintanence := FALSE;
   STATUS[483].EXT.Operation := FALSE;
   STATUS[483].EXT.Forced := FALSE;
   STATUS[483].EXT.BIT29 := FALSE;
   STATUS[483].EXT.BIT30 := FALSE;
   STATUS[483].EXT.BIT31 := FALSE;
   STATUS[483].EXT.ModeBit1 := FALSE;
   STATUS[483].EXT.ModeBit2 := FALSE;
   STATUS[483].EXT.ModeBit3 := FALSE;
   STATUS[483].EXT.BIT19 := FALSE;
   STATUS[483].EXT.BIT20 := FALSE;
   STATUS[483].EXT.AlarmSuppressed := FALSE;
   STATUS[483].EXT.AlarmPresent := FALSE;
   STATUS[483].EXT.AlarmFailUnAck := FALSE;
   STATUS[483].Status := 0;
   STATUS[483].TimeStamp := 16#0000;
   STATUS[484].EXT.AlarmWarnUnAck := FALSE;
   STATUS[484].EXT.AckRequired := FALSE;
   STATUS[484].EXT.Maintanence := FALSE;
   STATUS[484].EXT.Operation := FALSE;
   STATUS[484].EXT.Forced := FALSE;
   STATUS[484].EXT.BIT29 := FALSE;
   STATUS[484].EXT.BIT30 := FALSE;
   STATUS[484].EXT.BIT31 := FALSE;
   STATUS[484].EXT.ModeBit1 := FALSE;
   STATUS[484].EXT.ModeBit2 := FALSE;
   STATUS[484].EXT.ModeBit3 := FALSE;
   STATUS[484].EXT.BIT19 := FALSE;
   STATUS[484].EXT.BIT20 := FALSE;
   STATUS[484].EXT.AlarmSuppressed := FALSE;
   STATUS[484].EXT.AlarmPresent := FALSE;
   STATUS[484].EXT.AlarmFailUnAck := FALSE;
   STATUS[484].Status := 0;
   STATUS[484].TimeStamp := 16#0000;
   STATUS[485].EXT.AlarmWarnUnAck := FALSE;
   STATUS[485].EXT.AckRequired := FALSE;
   STATUS[485].EXT.Maintanence := FALSE;
   STATUS[485].EXT.Operation := FALSE;
   STATUS[485].EXT.Forced := FALSE;
   STATUS[485].EXT.BIT29 := FALSE;
   STATUS[485].EXT.BIT30 := FALSE;
   STATUS[485].EXT.BIT31 := FALSE;
   STATUS[485].EXT.ModeBit1 := FALSE;
   STATUS[485].EXT.ModeBit2 := FALSE;
   STATUS[485].EXT.ModeBit3 := FALSE;
   STATUS[485].EXT.BIT19 := FALSE;
   STATUS[485].EXT.BIT20 := FALSE;
   STATUS[485].EXT.AlarmSuppressed := FALSE;
   STATUS[485].EXT.AlarmPresent := FALSE;
   STATUS[485].EXT.AlarmFailUnAck := FALSE;
   STATUS[485].Status := 0;
   STATUS[485].TimeStamp := 16#0000;
   STATUS[486].EXT.AlarmWarnUnAck := FALSE;
   STATUS[486].EXT.AckRequired := FALSE;
   STATUS[486].EXT.Maintanence := FALSE;
   STATUS[486].EXT.Operation := FALSE;
   STATUS[486].EXT.Forced := FALSE;
   STATUS[486].EXT.BIT29 := FALSE;
   STATUS[486].EXT.BIT30 := FALSE;
   STATUS[486].EXT.BIT31 := FALSE;
   STATUS[486].EXT.ModeBit1 := FALSE;
   STATUS[486].EXT.ModeBit2 := FALSE;
   STATUS[486].EXT.ModeBit3 := FALSE;
   STATUS[486].EXT.BIT19 := FALSE;
   STATUS[486].EXT.BIT20 := FALSE;
   STATUS[486].EXT.AlarmSuppressed := FALSE;
   STATUS[486].EXT.AlarmPresent := FALSE;
   STATUS[486].EXT.AlarmFailUnAck := FALSE;
   STATUS[486].Status := 0;
   STATUS[486].TimeStamp := 16#0000;
   STATUS[487].EXT.AlarmWarnUnAck := FALSE;
   STATUS[487].EXT.AckRequired := FALSE;
   STATUS[487].EXT.Maintanence := FALSE;
   STATUS[487].EXT.Operation := FALSE;
   STATUS[487].EXT.Forced := FALSE;
   STATUS[487].EXT.BIT29 := FALSE;
   STATUS[487].EXT.BIT30 := FALSE;
   STATUS[487].EXT.BIT31 := FALSE;
   STATUS[487].EXT.ModeBit1 := FALSE;
   STATUS[487].EXT.ModeBit2 := FALSE;
   STATUS[487].EXT.ModeBit3 := FALSE;
   STATUS[487].EXT.BIT19 := FALSE;
   STATUS[487].EXT.BIT20 := FALSE;
   STATUS[487].EXT.AlarmSuppressed := FALSE;
   STATUS[487].EXT.AlarmPresent := FALSE;
   STATUS[487].EXT.AlarmFailUnAck := FALSE;
   STATUS[487].Status := 0;
   STATUS[487].TimeStamp := 16#0000;
   STATUS[488].EXT.AlarmWarnUnAck := FALSE;
   STATUS[488].EXT.AckRequired := FALSE;
   STATUS[488].EXT.Maintanence := FALSE;
   STATUS[488].EXT.Operation := FALSE;
   STATUS[488].EXT.Forced := FALSE;
   STATUS[488].EXT.BIT29 := FALSE;
   STATUS[488].EXT.BIT30 := FALSE;
   STATUS[488].EXT.BIT31 := FALSE;
   STATUS[488].EXT.ModeBit1 := FALSE;
   STATUS[488].EXT.ModeBit2 := FALSE;
   STATUS[488].EXT.ModeBit3 := FALSE;
   STATUS[488].EXT.BIT19 := FALSE;
   STATUS[488].EXT.BIT20 := FALSE;
   STATUS[488].EXT.AlarmSuppressed := FALSE;
   STATUS[488].EXT.AlarmPresent := FALSE;
   STATUS[488].EXT.AlarmFailUnAck := FALSE;
   STATUS[488].Status := 0;
   STATUS[488].TimeStamp := 16#0000;
   STATUS[489].EXT.AlarmWarnUnAck := FALSE;
   STATUS[489].EXT.AckRequired := FALSE;
   STATUS[489].EXT.Maintanence := FALSE;
   STATUS[489].EXT.Operation := FALSE;
   STATUS[489].EXT.Forced := FALSE;
   STATUS[489].EXT.BIT29 := FALSE;
   STATUS[489].EXT.BIT30 := FALSE;
   STATUS[489].EXT.BIT31 := FALSE;
   STATUS[489].EXT.ModeBit1 := FALSE;
   STATUS[489].EXT.ModeBit2 := FALSE;
   STATUS[489].EXT.ModeBit3 := FALSE;
   STATUS[489].EXT.BIT19 := FALSE;
   STATUS[489].EXT.BIT20 := FALSE;
   STATUS[489].EXT.AlarmSuppressed := FALSE;
   STATUS[489].EXT.AlarmPresent := FALSE;
   STATUS[489].EXT.AlarmFailUnAck := FALSE;
   STATUS[489].Status := 0;
   STATUS[489].TimeStamp := 16#0000;
   STATUS[490].EXT.AlarmWarnUnAck := FALSE;
   STATUS[490].EXT.AckRequired := FALSE;
   STATUS[490].EXT.Maintanence := FALSE;
   STATUS[490].EXT.Operation := FALSE;
   STATUS[490].EXT.Forced := FALSE;
   STATUS[490].EXT.BIT29 := FALSE;
   STATUS[490].EXT.BIT30 := FALSE;
   STATUS[490].EXT.BIT31 := FALSE;
   STATUS[490].EXT.ModeBit1 := FALSE;
   STATUS[490].EXT.ModeBit2 := FALSE;
   STATUS[490].EXT.ModeBit3 := FALSE;
   STATUS[490].EXT.BIT19 := FALSE;
   STATUS[490].EXT.BIT20 := FALSE;
   STATUS[490].EXT.AlarmSuppressed := FALSE;
   STATUS[490].EXT.AlarmPresent := FALSE;
   STATUS[490].EXT.AlarmFailUnAck := FALSE;
   STATUS[490].Status := 0;
   STATUS[490].TimeStamp := 16#0000;
   STATUS[491].EXT.AlarmWarnUnAck := FALSE;
   STATUS[491].EXT.AckRequired := FALSE;
   STATUS[491].EXT.Maintanence := FALSE;
   STATUS[491].EXT.Operation := FALSE;
   STATUS[491].EXT.Forced := FALSE;
   STATUS[491].EXT.BIT29 := FALSE;
   STATUS[491].EXT.BIT30 := FALSE;
   STATUS[491].EXT.BIT31 := FALSE;
   STATUS[491].EXT.ModeBit1 := FALSE;
   STATUS[491].EXT.ModeBit2 := FALSE;
   STATUS[491].EXT.ModeBit3 := FALSE;
   STATUS[491].EXT.BIT19 := FALSE;
   STATUS[491].EXT.BIT20 := FALSE;
   STATUS[491].EXT.AlarmSuppressed := FALSE;
   STATUS[491].EXT.AlarmPresent := FALSE;
   STATUS[491].EXT.AlarmFailUnAck := FALSE;
   STATUS[491].Status := 0;
   STATUS[491].TimeStamp := 16#0000;
   STATUS[492].EXT.AlarmWarnUnAck := FALSE;
   STATUS[492].EXT.AckRequired := FALSE;
   STATUS[492].EXT.Maintanence := FALSE;
   STATUS[492].EXT.Operation := FALSE;
   STATUS[492].EXT.Forced := FALSE;
   STATUS[492].EXT.BIT29 := FALSE;
   STATUS[492].EXT.BIT30 := FALSE;
   STATUS[492].EXT.BIT31 := FALSE;
   STATUS[492].EXT.ModeBit1 := FALSE;
   STATUS[492].EXT.ModeBit2 := FALSE;
   STATUS[492].EXT.ModeBit3 := FALSE;
   STATUS[492].EXT.BIT19 := FALSE;
   STATUS[492].EXT.BIT20 := FALSE;
   STATUS[492].EXT.AlarmSuppressed := FALSE;
   STATUS[492].EXT.AlarmPresent := FALSE;
   STATUS[492].EXT.AlarmFailUnAck := FALSE;
   STATUS[492].Status := 0;
   STATUS[492].TimeStamp := 16#0000;
   STATUS[493].EXT.AlarmWarnUnAck := FALSE;
   STATUS[493].EXT.AckRequired := FALSE;
   STATUS[493].EXT.Maintanence := FALSE;
   STATUS[493].EXT.Operation := FALSE;
   STATUS[493].EXT.Forced := FALSE;
   STATUS[493].EXT.BIT29 := FALSE;
   STATUS[493].EXT.BIT30 := FALSE;
   STATUS[493].EXT.BIT31 := FALSE;
   STATUS[493].EXT.ModeBit1 := FALSE;
   STATUS[493].EXT.ModeBit2 := FALSE;
   STATUS[493].EXT.ModeBit3 := FALSE;
   STATUS[493].EXT.BIT19 := FALSE;
   STATUS[493].EXT.BIT20 := FALSE;
   STATUS[493].EXT.AlarmSuppressed := FALSE;
   STATUS[493].EXT.AlarmPresent := FALSE;
   STATUS[493].EXT.AlarmFailUnAck := FALSE;
   STATUS[493].Status := 0;
   STATUS[493].TimeStamp := 16#0000;
   STATUS[494].EXT.AlarmWarnUnAck := FALSE;
   STATUS[494].EXT.AckRequired := FALSE;
   STATUS[494].EXT.Maintanence := FALSE;
   STATUS[494].EXT.Operation := FALSE;
   STATUS[494].EXT.Forced := FALSE;
   STATUS[494].EXT.BIT29 := FALSE;
   STATUS[494].EXT.BIT30 := FALSE;
   STATUS[494].EXT.BIT31 := FALSE;
   STATUS[494].EXT.ModeBit1 := FALSE;
   STATUS[494].EXT.ModeBit2 := FALSE;
   STATUS[494].EXT.ModeBit3 := FALSE;
   STATUS[494].EXT.BIT19 := FALSE;
   STATUS[494].EXT.BIT20 := FALSE;
   STATUS[494].EXT.AlarmSuppressed := FALSE;
   STATUS[494].EXT.AlarmPresent := FALSE;
   STATUS[494].EXT.AlarmFailUnAck := FALSE;
   STATUS[494].Status := 0;
   STATUS[494].TimeStamp := 16#0000;
   STATUS[495].EXT.AlarmWarnUnAck := FALSE;
   STATUS[495].EXT.AckRequired := FALSE;
   STATUS[495].EXT.Maintanence := FALSE;
   STATUS[495].EXT.Operation := FALSE;
   STATUS[495].EXT.Forced := FALSE;
   STATUS[495].EXT.BIT29 := FALSE;
   STATUS[495].EXT.BIT30 := FALSE;
   STATUS[495].EXT.BIT31 := FALSE;
   STATUS[495].EXT.ModeBit1 := FALSE;
   STATUS[495].EXT.ModeBit2 := FALSE;
   STATUS[495].EXT.ModeBit3 := FALSE;
   STATUS[495].EXT.BIT19 := FALSE;
   STATUS[495].EXT.BIT20 := FALSE;
   STATUS[495].EXT.AlarmSuppressed := FALSE;
   STATUS[495].EXT.AlarmPresent := FALSE;
   STATUS[495].EXT.AlarmFailUnAck := FALSE;
   STATUS[495].Status := 0;
   STATUS[495].TimeStamp := 16#0000;
   STATUS[496].EXT.AlarmWarnUnAck := FALSE;
   STATUS[496].EXT.AckRequired := FALSE;
   STATUS[496].EXT.Maintanence := FALSE;
   STATUS[496].EXT.Operation := FALSE;
   STATUS[496].EXT.Forced := FALSE;
   STATUS[496].EXT.BIT29 := FALSE;
   STATUS[496].EXT.BIT30 := FALSE;
   STATUS[496].EXT.BIT31 := FALSE;
   STATUS[496].EXT.ModeBit1 := FALSE;
   STATUS[496].EXT.ModeBit2 := FALSE;
   STATUS[496].EXT.ModeBit3 := FALSE;
   STATUS[496].EXT.BIT19 := FALSE;
   STATUS[496].EXT.BIT20 := FALSE;
   STATUS[496].EXT.AlarmSuppressed := FALSE;
   STATUS[496].EXT.AlarmPresent := FALSE;
   STATUS[496].EXT.AlarmFailUnAck := FALSE;
   STATUS[496].Status := 0;
   STATUS[496].TimeStamp := 16#0000;
   STATUS[497].EXT.AlarmWarnUnAck := FALSE;
   STATUS[497].EXT.AckRequired := FALSE;
   STATUS[497].EXT.Maintanence := FALSE;
   STATUS[497].EXT.Operation := FALSE;
   STATUS[497].EXT.Forced := FALSE;
   STATUS[497].EXT.BIT29 := FALSE;
   STATUS[497].EXT.BIT30 := FALSE;
   STATUS[497].EXT.BIT31 := FALSE;
   STATUS[497].EXT.ModeBit1 := FALSE;
   STATUS[497].EXT.ModeBit2 := FALSE;
   STATUS[497].EXT.ModeBit3 := FALSE;
   STATUS[497].EXT.BIT19 := FALSE;
   STATUS[497].EXT.BIT20 := FALSE;
   STATUS[497].EXT.AlarmSuppressed := FALSE;
   STATUS[497].EXT.AlarmPresent := FALSE;
   STATUS[497].EXT.AlarmFailUnAck := FALSE;
   STATUS[497].Status := 0;
   STATUS[497].TimeStamp := 16#0000;
   STATUS[498].EXT.AlarmWarnUnAck := FALSE;
   STATUS[498].EXT.AckRequired := FALSE;
   STATUS[498].EXT.Maintanence := FALSE;
   STATUS[498].EXT.Operation := FALSE;
   STATUS[498].EXT.Forced := FALSE;
   STATUS[498].EXT.BIT29 := FALSE;
   STATUS[498].EXT.BIT30 := FALSE;
   STATUS[498].EXT.BIT31 := FALSE;
   STATUS[498].EXT.ModeBit1 := FALSE;
   STATUS[498].EXT.ModeBit2 := FALSE;
   STATUS[498].EXT.ModeBit3 := FALSE;
   STATUS[498].EXT.BIT19 := FALSE;
   STATUS[498].EXT.BIT20 := FALSE;
   STATUS[498].EXT.AlarmSuppressed := FALSE;
   STATUS[498].EXT.AlarmPresent := FALSE;
   STATUS[498].EXT.AlarmFailUnAck := FALSE;
   STATUS[498].Status := 0;
   STATUS[498].TimeStamp := 16#0000;
   STATUS[499].EXT.AlarmWarnUnAck := FALSE;
   STATUS[499].EXT.AckRequired := FALSE;
   STATUS[499].EXT.Maintanence := FALSE;
   STATUS[499].EXT.Operation := FALSE;
   STATUS[499].EXT.Forced := FALSE;
   STATUS[499].EXT.BIT29 := FALSE;
   STATUS[499].EXT.BIT30 := FALSE;
   STATUS[499].EXT.BIT31 := FALSE;
   STATUS[499].EXT.ModeBit1 := FALSE;
   STATUS[499].EXT.ModeBit2 := FALSE;
   STATUS[499].EXT.ModeBit3 := FALSE;
   STATUS[499].EXT.BIT19 := FALSE;
   STATUS[499].EXT.BIT20 := FALSE;
   STATUS[499].EXT.AlarmSuppressed := FALSE;
   STATUS[499].EXT.AlarmPresent := FALSE;
   STATUS[499].EXT.AlarmFailUnAck := FALSE;
   STATUS[499].Status := 0;
   STATUS[499].TimeStamp := 16#0000;
   STATUS[500].EXT.AlarmWarnUnAck := FALSE;
   STATUS[500].EXT.AckRequired := FALSE;
   STATUS[500].EXT.Maintanence := FALSE;
   STATUS[500].EXT.Operation := FALSE;
   STATUS[500].EXT.Forced := FALSE;
   STATUS[500].EXT.BIT29 := FALSE;
   STATUS[500].EXT.BIT30 := FALSE;
   STATUS[500].EXT.BIT31 := FALSE;
   STATUS[500].EXT.ModeBit1 := FALSE;
   STATUS[500].EXT.ModeBit2 := FALSE;
   STATUS[500].EXT.ModeBit3 := FALSE;
   STATUS[500].EXT.BIT19 := FALSE;
   STATUS[500].EXT.BIT20 := FALSE;
   STATUS[500].EXT.AlarmSuppressed := FALSE;
   STATUS[500].EXT.AlarmPresent := FALSE;
   STATUS[500].EXT.AlarmFailUnAck := FALSE;
   STATUS[500].Status := 0;
   STATUS[500].TimeStamp := 16#0000;
END_DATA_BLOCK

DATA_BLOCK "art_test_db"   // DB3
{ S7_Optimized_Access := 'FALSE' }
VERSION : 0.1
   VAR
      "bool" : Bool := FALSE;
      bool_47 : Bool := FALSE;
      bool_46 : Bool := FALSE;
      bool_45 : Bool := FALSE;
      bool_44 : Bool := FALSE;
      bool_43 : Bool := FALSE;
      bool_42 : Bool := FALSE;
      bool_41 : Bool := FALSE;
      bool_40 : Bool := FALSE;
      bool_39 : Bool := FALSE;
      bool_38 : Bool := FALSE;
      bool_37 : Bool := FALSE;
      bool_36 : Bool := FALSE;
      bool_35 : Bool := FALSE;
      bool_34 : Bool := FALSE;
      bool_33 : Bool := FALSE;
      bool_32 : Bool := FALSE;
      bool_31 : Bool := FALSE;
      bool_30 : Bool := FALSE;
      bool_29 : Bool := FALSE;
      bool_28 : Bool := FALSE;
      bool_27 : Bool := FALSE;
      bool_26 : Bool := FALSE;
      bool_25 : Bool := FALSE;
      bool_24 : Bool := FALSE;
      bool_23 : Bool := FALSE;
      bool_22 : Bool := FALSE;
      bool_21 : Bool := FALSE;
      bool_20 : Bool := FALSE;
      bool_19 : Bool := FALSE;
      bool_18 : Bool := FALSE;
      bool_17 : Bool := FALSE;
      bool_16 : Bool := FALSE;
      bool_15 : Bool := FALSE;
      bool_14 : Bool := FALSE;
      bool_13 : Bool := FALSE;
      bool_12 : Bool := FALSE;
      bool_11 : Bool := FALSE;
      bool_10 : Bool := FALSE;
      bool_9 : Bool := FALSE;
      bool_8 : Bool := FALSE;
      bool_7 : Bool := FALSE;
      bool_6 : Bool := FALSE;
      bool_5 : Bool := FALSE;
      bool_4 : Bool := FALSE;
      bool_3 : Bool := FALSE;
      bool_2 : Bool := FALSE;
      bool_1 : Bool := FALSE;
      bool2 : Bool := FALSE;
   END_VAR
BEGIN
END_DATA_BLOCK

DATA_BLOCK "ACESYS_HMI_UNIT"   // DB4
TITLE = ACESYS UNIT DB
{ S7_Optimized_Access := 'FALSE' }
AUTHOR : METIS
FAMILY : ACESYS
NAME : UnitDB
VERSION : 8.0
   VAR
      STATUS : Array[0..1000] of "ACESYS_HMI_STAT_32T";   // Unit Status to HMI
   END_VAR
BEGIN
   STATUS[0].EXT.AlarmWarnUnAck := FALSE;
   STATUS[0].EXT.AckRequired := FALSE;
   STATUS[0].EXT.Maintanence := FALSE;
   STATUS[0].EXT.Operation := FALSE;
   STATUS[0].EXT.Forced := FALSE;
   STATUS[0].EXT.BIT29 := FALSE;
   STATUS[0].EXT.BIT30 := FALSE;
   STATUS[0].EXT.BIT31 := FALSE;
   STATUS[0].EXT.ModeBit1 := FALSE;
   STATUS[0].EXT.ModeBit2 := FALSE;
   STATUS[0].EXT.ModeBit3 := FALSE;
   STATUS[0].EXT.BIT19 := FALSE;
   STATUS[0].EXT.BIT20 := FALSE;
   STATUS[0].EXT.AlarmSuppressed := FALSE;
   STATUS[0].EXT.AlarmPresent := FALSE;
   STATUS[0].EXT.AlarmFailUnAck := FALSE;
   STATUS[0].Status := 0;
   STATUS[0].TimeStamp := 16#0000;
   STATUS[1].EXT.AlarmWarnUnAck := FALSE;
   STATUS[1].EXT.AckRequired := FALSE;
   STATUS[1].EXT.Maintanence := FALSE;
   STATUS[1].EXT.Operation := FALSE;
   STATUS[1].EXT.Forced := FALSE;
   STATUS[1].EXT.BIT29 := FALSE;
   STATUS[1].EXT.BIT30 := FALSE;
   STATUS[1].EXT.BIT31 := FALSE;
   STATUS[1].EXT.ModeBit1 := FALSE;
   STATUS[1].EXT.ModeBit2 := FALSE;
   STATUS[1].EXT.ModeBit3 := FALSE;
   STATUS[1].EXT.BIT19 := FALSE;
   STATUS[1].EXT.BIT20 := FALSE;
   STATUS[1].EXT.AlarmSuppressed := FALSE;
   STATUS[1].EXT.AlarmPresent := TRUE;
   STATUS[1].EXT.AlarmFailUnAck := FALSE;
   STATUS[1].Status := 1;
   STATUS[1].TimeStamp := 16#3928;
   STATUS[2].EXT.AlarmWarnUnAck := FALSE;
   STATUS[2].EXT.AckRequired := FALSE;
   STATUS[2].EXT.Maintanence := FALSE;
   STATUS[2].EXT.Operation := FALSE;
   STATUS[2].EXT.Forced := FALSE;
   STATUS[2].EXT.BIT29 := FALSE;
   STATUS[2].EXT.BIT30 := FALSE;
   STATUS[2].EXT.BIT31 := FALSE;
   STATUS[2].EXT.ModeBit1 := FALSE;
   STATUS[2].EXT.ModeBit2 := FALSE;
   STATUS[2].EXT.ModeBit3 := FALSE;
   STATUS[2].EXT.BIT19 := FALSE;
   STATUS[2].EXT.BIT20 := FALSE;
   STATUS[2].EXT.AlarmSuppressed := FALSE;
   STATUS[2].EXT.AlarmPresent := TRUE;
   STATUS[2].EXT.AlarmFailUnAck := TRUE;
   STATUS[2].Status := 121;
   STATUS[2].TimeStamp := 16#45F7;
   STATUS[3].EXT.AlarmWarnUnAck := FALSE;
   STATUS[3].EXT.AckRequired := FALSE;
   STATUS[3].EXT.Maintanence := FALSE;
   STATUS[3].EXT.Operation := FALSE;
   STATUS[3].EXT.Forced := FALSE;
   STATUS[3].EXT.BIT29 := FALSE;
   STATUS[3].EXT.BIT30 := FALSE;
   STATUS[3].EXT.BIT31 := FALSE;
   STATUS[3].EXT.ModeBit1 := FALSE;
   STATUS[3].EXT.ModeBit2 := FALSE;
   STATUS[3].EXT.ModeBit3 := FALSE;
   STATUS[3].EXT.BIT19 := FALSE;
   STATUS[3].EXT.BIT20 := FALSE;
   STATUS[3].EXT.AlarmSuppressed := FALSE;
   STATUS[3].EXT.AlarmPresent := TRUE;
   STATUS[3].EXT.AlarmFailUnAck := TRUE;
   STATUS[3].Status := 104;
   STATUS[3].TimeStamp := 16#3928;
   STATUS[4].EXT.AlarmWarnUnAck := FALSE;
   STATUS[4].EXT.AckRequired := FALSE;
   STATUS[4].EXT.Maintanence := FALSE;
   STATUS[4].EXT.Operation := FALSE;
   STATUS[4].EXT.Forced := FALSE;
   STATUS[4].EXT.BIT29 := FALSE;
   STATUS[4].EXT.BIT30 := FALSE;
   STATUS[4].EXT.BIT31 := FALSE;
   STATUS[4].EXT.ModeBit1 := FALSE;
   STATUS[4].EXT.ModeBit2 := FALSE;
   STATUS[4].EXT.ModeBit3 := FALSE;
   STATUS[4].EXT.BIT19 := FALSE;
   STATUS[4].EXT.BIT20 := FALSE;
   STATUS[4].EXT.AlarmSuppressed := FALSE;
   STATUS[4].EXT.AlarmPresent := TRUE;
   STATUS[4].EXT.AlarmFailUnAck := TRUE;
   STATUS[4].Status := 105;
   STATUS[4].TimeStamp := 16#3928;
   STATUS[5].EXT.AlarmWarnUnAck := FALSE;
   STATUS[5].EXT.AckRequired := FALSE;
   STATUS[5].EXT.Maintanence := FALSE;
   STATUS[5].EXT.Operation := FALSE;
   STATUS[5].EXT.Forced := FALSE;
   STATUS[5].EXT.BIT29 := FALSE;
   STATUS[5].EXT.BIT30 := FALSE;
   STATUS[5].EXT.BIT31 := FALSE;
   STATUS[5].EXT.ModeBit1 := FALSE;
   STATUS[5].EXT.ModeBit2 := FALSE;
   STATUS[5].EXT.ModeBit3 := FALSE;
   STATUS[5].EXT.BIT19 := FALSE;
   STATUS[5].EXT.BIT20 := FALSE;
   STATUS[5].EXT.AlarmSuppressed := FALSE;
   STATUS[5].EXT.AlarmPresent := TRUE;
   STATUS[5].EXT.AlarmFailUnAck := TRUE;
   STATUS[5].Status := 104;
   STATUS[5].TimeStamp := 16#3928;
   STATUS[6].EXT.AlarmWarnUnAck := FALSE;
   STATUS[6].EXT.AckRequired := TRUE;
   STATUS[6].EXT.Maintanence := FALSE;
   STATUS[6].EXT.Operation := TRUE;
   STATUS[6].EXT.Forced := FALSE;
   STATUS[6].EXT.BIT29 := FALSE;
   STATUS[6].EXT.BIT30 := FALSE;
   STATUS[6].EXT.BIT31 := FALSE;
   STATUS[6].EXT.ModeBit1 := FALSE;
   STATUS[6].EXT.ModeBit2 := FALSE;
   STATUS[6].EXT.ModeBit3 := FALSE;
   STATUS[6].EXT.BIT19 := FALSE;
   STATUS[6].EXT.BIT20 := FALSE;
   STATUS[6].EXT.AlarmSuppressed := FALSE;
   STATUS[6].EXT.AlarmPresent := FALSE;
   STATUS[6].EXT.AlarmFailUnAck := TRUE;
   STATUS[6].Status := 10;
   STATUS[6].TimeStamp := 16#84BA;
   STATUS[7].EXT.AlarmWarnUnAck := FALSE;
   STATUS[7].EXT.AckRequired := TRUE;
   STATUS[7].EXT.Maintanence := FALSE;
   STATUS[7].EXT.Operation := TRUE;
   STATUS[7].EXT.Forced := FALSE;
   STATUS[7].EXT.BIT29 := FALSE;
   STATUS[7].EXT.BIT30 := FALSE;
   STATUS[7].EXT.BIT31 := FALSE;
   STATUS[7].EXT.ModeBit1 := FALSE;
   STATUS[7].EXT.ModeBit2 := FALSE;
   STATUS[7].EXT.ModeBit3 := FALSE;
   STATUS[7].EXT.BIT19 := FALSE;
   STATUS[7].EXT.BIT20 := FALSE;
   STATUS[7].EXT.AlarmSuppressed := FALSE;
   STATUS[7].EXT.AlarmPresent := FALSE;
   STATUS[7].EXT.AlarmFailUnAck := TRUE;
   STATUS[7].Status := 10;
   STATUS[7].TimeStamp := 16#84BA;
   STATUS[8].EXT.AlarmWarnUnAck := FALSE;
   STATUS[8].EXT.AckRequired := FALSE;
   STATUS[8].EXT.Maintanence := FALSE;
   STATUS[8].EXT.Operation := FALSE;
   STATUS[8].EXT.Forced := FALSE;
   STATUS[8].EXT.BIT29 := FALSE;
   STATUS[8].EXT.BIT30 := FALSE;
   STATUS[8].EXT.BIT31 := FALSE;
   STATUS[8].EXT.ModeBit1 := FALSE;
   STATUS[8].EXT.ModeBit2 := FALSE;
   STATUS[8].EXT.ModeBit3 := FALSE;
   STATUS[8].EXT.BIT19 := FALSE;
   STATUS[8].EXT.BIT20 := FALSE;
   STATUS[8].EXT.AlarmSuppressed := FALSE;
   STATUS[8].EXT.AlarmPresent := FALSE;
   STATUS[8].EXT.AlarmFailUnAck := FALSE;
   STATUS[8].Status := 1;
   STATUS[8].TimeStamp := 16#E770;
   STATUS[9].EXT.AlarmWarnUnAck := FALSE;
   STATUS[9].EXT.AckRequired := FALSE;
   STATUS[9].EXT.Maintanence := FALSE;
   STATUS[9].EXT.Operation := FALSE;
   STATUS[9].EXT.Forced := FALSE;
   STATUS[9].EXT.BIT29 := FALSE;
   STATUS[9].EXT.BIT30 := FALSE;
   STATUS[9].EXT.BIT31 := FALSE;
   STATUS[9].EXT.ModeBit1 := FALSE;
   STATUS[9].EXT.ModeBit2 := FALSE;
   STATUS[9].EXT.ModeBit3 := FALSE;
   STATUS[9].EXT.BIT19 := FALSE;
   STATUS[9].EXT.BIT20 := FALSE;
   STATUS[9].EXT.AlarmSuppressed := FALSE;
   STATUS[9].EXT.AlarmPresent := FALSE;
   STATUS[9].EXT.AlarmFailUnAck := FALSE;
   STATUS[9].Status := 1;
   STATUS[9].TimeStamp := 16#E6A1;
   STATUS[10].EXT.AlarmWarnUnAck := FALSE;
   STATUS[10].EXT.AckRequired := FALSE;
   STATUS[10].EXT.Maintanence := FALSE;
   STATUS[10].EXT.Operation := FALSE;
   STATUS[10].EXT.Forced := FALSE;
   STATUS[10].EXT.BIT29 := FALSE;
   STATUS[10].EXT.BIT30 := FALSE;
   STATUS[10].EXT.BIT31 := FALSE;
   STATUS[10].EXT.ModeBit1 := FALSE;
   STATUS[10].EXT.ModeBit2 := FALSE;
   STATUS[10].EXT.ModeBit3 := FALSE;
   STATUS[10].EXT.BIT19 := FALSE;
   STATUS[10].EXT.BIT20 := FALSE;
   STATUS[10].EXT.AlarmSuppressed := FALSE;
   STATUS[10].EXT.AlarmPresent := FALSE;
   STATUS[10].EXT.AlarmFailUnAck := FALSE;
   STATUS[10].Status := 1;
   STATUS[10].TimeStamp := 16#E688;
   STATUS[11].EXT.AlarmWarnUnAck := FALSE;
   STATUS[11].EXT.AckRequired := FALSE;
   STATUS[11].EXT.Maintanence := FALSE;
   STATUS[11].EXT.Operation := FALSE;
   STATUS[11].EXT.Forced := FALSE;
   STATUS[11].EXT.BIT29 := FALSE;
   STATUS[11].EXT.BIT30 := FALSE;
   STATUS[11].EXT.BIT31 := FALSE;
   STATUS[11].EXT.ModeBit1 := FALSE;
   STATUS[11].EXT.ModeBit2 := FALSE;
   STATUS[11].EXT.ModeBit3 := FALSE;
   STATUS[11].EXT.BIT19 := FALSE;
   STATUS[11].EXT.BIT20 := FALSE;
   STATUS[11].EXT.AlarmSuppressed := FALSE;
   STATUS[11].EXT.AlarmPresent := FALSE;
   STATUS[11].EXT.AlarmFailUnAck := FALSE;
   STATUS[11].Status := 1;
   STATUS[11].TimeStamp := 16#E694;
   STATUS[12].EXT.AlarmWarnUnAck := FALSE;
   STATUS[12].EXT.AckRequired := FALSE;
   STATUS[12].EXT.Maintanence := FALSE;
   STATUS[12].EXT.Operation := FALSE;
   STATUS[12].EXT.Forced := FALSE;
   STATUS[12].EXT.BIT29 := FALSE;
   STATUS[12].EXT.BIT30 := FALSE;
   STATUS[12].EXT.BIT31 := FALSE;
   STATUS[12].EXT.ModeBit1 := FALSE;
   STATUS[12].EXT.ModeBit2 := FALSE;
   STATUS[12].EXT.ModeBit3 := FALSE;
   STATUS[12].EXT.BIT19 := FALSE;
   STATUS[12].EXT.BIT20 := FALSE;
   STATUS[12].EXT.AlarmSuppressed := FALSE;
   STATUS[12].EXT.AlarmPresent := FALSE;
   STATUS[12].EXT.AlarmFailUnAck := FALSE;
   STATUS[12].Status := 1;
   STATUS[12].TimeStamp := 16#E694;
   STATUS[13].EXT.AlarmWarnUnAck := FALSE;
   STATUS[13].EXT.AckRequired := FALSE;
   STATUS[13].EXT.Maintanence := FALSE;
   STATUS[13].EXT.Operation := FALSE;
   STATUS[13].EXT.Forced := FALSE;
   STATUS[13].EXT.BIT29 := FALSE;
   STATUS[13].EXT.BIT30 := FALSE;
   STATUS[13].EXT.BIT31 := FALSE;
   STATUS[13].EXT.ModeBit1 := FALSE;
   STATUS[13].EXT.ModeBit2 := FALSE;
   STATUS[13].EXT.ModeBit3 := FALSE;
   STATUS[13].EXT.BIT19 := FALSE;
   STATUS[13].EXT.BIT20 := FALSE;
   STATUS[13].EXT.AlarmSuppressed := FALSE;
   STATUS[13].EXT.AlarmPresent := FALSE;
   STATUS[13].EXT.AlarmFailUnAck := FALSE;
   STATUS[13].Status := 1;
   STATUS[13].TimeStamp := 16#E694;
   STATUS[14].EXT.AlarmWarnUnAck := FALSE;
   STATUS[14].EXT.AckRequired := FALSE;
   STATUS[14].EXT.Maintanence := FALSE;
   STATUS[14].EXT.Operation := FALSE;
   STATUS[14].EXT.Forced := FALSE;
   STATUS[14].EXT.BIT29 := FALSE;
   STATUS[14].EXT.BIT30 := FALSE;
   STATUS[14].EXT.BIT31 := FALSE;
   STATUS[14].EXT.ModeBit1 := FALSE;
   STATUS[14].EXT.ModeBit2 := FALSE;
   STATUS[14].EXT.ModeBit3 := FALSE;
   STATUS[14].EXT.BIT19 := FALSE;
   STATUS[14].EXT.BIT20 := FALSE;
   STATUS[14].EXT.AlarmSuppressed := TRUE;
   STATUS[14].EXT.AlarmPresent := FALSE;
   STATUS[14].EXT.AlarmFailUnAck := FALSE;
   STATUS[14].Status := 1;
   STATUS[14].TimeStamp := 16#35D8;
   STATUS[15].EXT.AlarmWarnUnAck := FALSE;
   STATUS[15].EXT.AckRequired := FALSE;
   STATUS[15].EXT.Maintanence := FALSE;
   STATUS[15].EXT.Operation := FALSE;
   STATUS[15].EXT.Forced := FALSE;
   STATUS[15].EXT.BIT29 := FALSE;
   STATUS[15].EXT.BIT30 := FALSE;
   STATUS[15].EXT.BIT31 := FALSE;
   STATUS[15].EXT.ModeBit1 := FALSE;
   STATUS[15].EXT.ModeBit2 := FALSE;
   STATUS[15].EXT.ModeBit3 := FALSE;
   STATUS[15].EXT.BIT19 := FALSE;
   STATUS[15].EXT.BIT20 := FALSE;
   STATUS[15].EXT.AlarmSuppressed := FALSE;
   STATUS[15].EXT.AlarmPresent := FALSE;
   STATUS[15].EXT.AlarmFailUnAck := FALSE;
   STATUS[15].Status := -22466;
   STATUS[15].TimeStamp := 16#84BA;
   STATUS[16].EXT.AlarmWarnUnAck := FALSE;
   STATUS[16].EXT.AckRequired := FALSE;
   STATUS[16].EXT.Maintanence := FALSE;
   STATUS[16].EXT.Operation := FALSE;
   STATUS[16].EXT.Forced := TRUE;
   STATUS[16].EXT.BIT29 := FALSE;
   STATUS[16].EXT.BIT30 := FALSE;
   STATUS[16].EXT.BIT31 := FALSE;
   STATUS[16].EXT.ModeBit1 := FALSE;
   STATUS[16].EXT.ModeBit2 := FALSE;
   STATUS[16].EXT.ModeBit3 := FALSE;
   STATUS[16].EXT.BIT19 := FALSE;
   STATUS[16].EXT.BIT20 := FALSE;
   STATUS[16].EXT.AlarmSuppressed := TRUE;
   STATUS[16].EXT.AlarmPresent := TRUE;
   STATUS[16].EXT.AlarmFailUnAck := TRUE;
   STATUS[16].Status := 190;
   STATUS[16].TimeStamp := 16#E0ED;
   STATUS[17].EXT.AlarmWarnUnAck := FALSE;
   STATUS[17].EXT.AckRequired := FALSE;
   STATUS[17].EXT.Maintanence := FALSE;
   STATUS[17].EXT.Operation := FALSE;
   STATUS[17].EXT.Forced := TRUE;
   STATUS[17].EXT.BIT29 := FALSE;
   STATUS[17].EXT.BIT30 := FALSE;
   STATUS[17].EXT.BIT31 := FALSE;
   STATUS[17].EXT.ModeBit1 := FALSE;
   STATUS[17].EXT.ModeBit2 := FALSE;
   STATUS[17].EXT.ModeBit3 := FALSE;
   STATUS[17].EXT.BIT19 := FALSE;
   STATUS[17].EXT.BIT20 := FALSE;
   STATUS[17].EXT.AlarmSuppressed := FALSE;
   STATUS[17].EXT.AlarmPresent := FALSE;
   STATUS[17].EXT.AlarmFailUnAck := TRUE;
   STATUS[17].Status := 190;
   STATUS[17].TimeStamp := 16#645C;
   STATUS[18].EXT.AlarmWarnUnAck := FALSE;
   STATUS[18].EXT.AckRequired := FALSE;
   STATUS[18].EXT.Maintanence := FALSE;
   STATUS[18].EXT.Operation := FALSE;
   STATUS[18].EXT.Forced := TRUE;
   STATUS[18].EXT.BIT29 := FALSE;
   STATUS[18].EXT.BIT30 := FALSE;
   STATUS[18].EXT.BIT31 := FALSE;
   STATUS[18].EXT.ModeBit1 := FALSE;
   STATUS[18].EXT.ModeBit2 := FALSE;
   STATUS[18].EXT.ModeBit3 := FALSE;
   STATUS[18].EXT.BIT19 := FALSE;
   STATUS[18].EXT.BIT20 := FALSE;
   STATUS[18].EXT.AlarmSuppressed := FALSE;
   STATUS[18].EXT.AlarmPresent := FALSE;
   STATUS[18].EXT.AlarmFailUnAck := TRUE;
   STATUS[18].Status := 190;
   STATUS[18].TimeStamp := 16#6A5C;
   STATUS[19].EXT.AlarmWarnUnAck := FALSE;
   STATUS[19].EXT.AckRequired := FALSE;
   STATUS[19].EXT.Maintanence := FALSE;
   STATUS[19].EXT.Operation := FALSE;
   STATUS[19].EXT.Forced := TRUE;
   STATUS[19].EXT.BIT29 := FALSE;
   STATUS[19].EXT.BIT30 := FALSE;
   STATUS[19].EXT.BIT31 := FALSE;
   STATUS[19].EXT.ModeBit1 := FALSE;
   STATUS[19].EXT.ModeBit2 := FALSE;
   STATUS[19].EXT.ModeBit3 := FALSE;
   STATUS[19].EXT.BIT19 := FALSE;
   STATUS[19].EXT.BIT20 := FALSE;
   STATUS[19].EXT.AlarmSuppressed := FALSE;
   STATUS[19].EXT.AlarmPresent := FALSE;
   STATUS[19].EXT.AlarmFailUnAck := TRUE;
   STATUS[19].Status := 190;
   STATUS[19].TimeStamp := 16#9BB3;
   STATUS[20].EXT.AlarmWarnUnAck := FALSE;
   STATUS[20].EXT.AckRequired := FALSE;
   STATUS[20].EXT.Maintanence := FALSE;
   STATUS[20].EXT.Operation := FALSE;
   STATUS[20].EXT.Forced := TRUE;
   STATUS[20].EXT.BIT29 := FALSE;
   STATUS[20].EXT.BIT30 := FALSE;
   STATUS[20].EXT.BIT31 := FALSE;
   STATUS[20].EXT.ModeBit1 := FALSE;
   STATUS[20].EXT.ModeBit2 := FALSE;
   STATUS[20].EXT.ModeBit3 := FALSE;
   STATUS[20].EXT.BIT19 := FALSE;
   STATUS[20].EXT.BIT20 := FALSE;
   STATUS[20].EXT.AlarmSuppressed := FALSE;
   STATUS[20].EXT.AlarmPresent := TRUE;
   STATUS[20].EXT.AlarmFailUnAck := TRUE;
   STATUS[20].Status := 190;
   STATUS[20].TimeStamp := 16#E973;
   STATUS[21].EXT.AlarmWarnUnAck := FALSE;
   STATUS[21].EXT.AckRequired := FALSE;
   STATUS[21].EXT.Maintanence := FALSE;
   STATUS[21].EXT.Operation := FALSE;
   STATUS[21].EXT.Forced := TRUE;
   STATUS[21].EXT.BIT29 := FALSE;
   STATUS[21].EXT.BIT30 := FALSE;
   STATUS[21].EXT.BIT31 := FALSE;
   STATUS[21].EXT.ModeBit1 := FALSE;
   STATUS[21].EXT.ModeBit2 := FALSE;
   STATUS[21].EXT.ModeBit3 := FALSE;
   STATUS[21].EXT.BIT19 := FALSE;
   STATUS[21].EXT.BIT20 := FALSE;
   STATUS[21].EXT.AlarmSuppressed := FALSE;
   STATUS[21].EXT.AlarmPresent := FALSE;
   STATUS[21].EXT.AlarmFailUnAck := TRUE;
   STATUS[21].Status := 190;
   STATUS[21].TimeStamp := 16#6EFC;
   STATUS[22].EXT.AlarmWarnUnAck := FALSE;
   STATUS[22].EXT.AckRequired := FALSE;
   STATUS[22].EXT.Maintanence := FALSE;
   STATUS[22].EXT.Operation := FALSE;
   STATUS[22].EXT.Forced := TRUE;
   STATUS[22].EXT.BIT29 := FALSE;
   STATUS[22].EXT.BIT30 := FALSE;
   STATUS[22].EXT.BIT31 := FALSE;
   STATUS[22].EXT.ModeBit1 := FALSE;
   STATUS[22].EXT.ModeBit2 := FALSE;
   STATUS[22].EXT.ModeBit3 := FALSE;
   STATUS[22].EXT.BIT19 := FALSE;
   STATUS[22].EXT.BIT20 := FALSE;
   STATUS[22].EXT.AlarmSuppressed := FALSE;
   STATUS[22].EXT.AlarmPresent := FALSE;
   STATUS[22].EXT.AlarmFailUnAck := TRUE;
   STATUS[22].Status := 190;
   STATUS[22].TimeStamp := 16#5BEC;
   STATUS[23].EXT.AlarmWarnUnAck := FALSE;
   STATUS[23].EXT.AckRequired := FALSE;
   STATUS[23].EXT.Maintanence := FALSE;
   STATUS[23].EXT.Operation := FALSE;
   STATUS[23].EXT.Forced := TRUE;
   STATUS[23].EXT.BIT29 := FALSE;
   STATUS[23].EXT.BIT30 := FALSE;
   STATUS[23].EXT.BIT31 := FALSE;
   STATUS[23].EXT.ModeBit1 := FALSE;
   STATUS[23].EXT.ModeBit2 := FALSE;
   STATUS[23].EXT.ModeBit3 := FALSE;
   STATUS[23].EXT.BIT19 := FALSE;
   STATUS[23].EXT.BIT20 := FALSE;
   STATUS[23].EXT.AlarmSuppressed := FALSE;
   STATUS[23].EXT.AlarmPresent := FALSE;
   STATUS[23].EXT.AlarmFailUnAck := TRUE;
   STATUS[23].Status := 190;
   STATUS[23].TimeStamp := 16#57A9;
   STATUS[24].EXT.AlarmWarnUnAck := FALSE;
   STATUS[24].EXT.AckRequired := FALSE;
   STATUS[24].EXT.Maintanence := FALSE;
   STATUS[24].EXT.Operation := FALSE;
   STATUS[24].EXT.Forced := TRUE;
   STATUS[24].EXT.BIT29 := FALSE;
   STATUS[24].EXT.BIT30 := FALSE;
   STATUS[24].EXT.BIT31 := FALSE;
   STATUS[24].EXT.ModeBit1 := FALSE;
   STATUS[24].EXT.ModeBit2 := FALSE;
   STATUS[24].EXT.ModeBit3 := FALSE;
   STATUS[24].EXT.BIT19 := FALSE;
   STATUS[24].EXT.BIT20 := FALSE;
   STATUS[24].EXT.AlarmSuppressed := FALSE;
   STATUS[24].EXT.AlarmPresent := FALSE;
   STATUS[24].EXT.AlarmFailUnAck := TRUE;
   STATUS[24].Status := 190;
   STATUS[24].TimeStamp := 16#5F8B;
   STATUS[25].EXT.AlarmWarnUnAck := FALSE;
   STATUS[25].EXT.AckRequired := FALSE;
   STATUS[25].EXT.Maintanence := FALSE;
   STATUS[25].EXT.Operation := FALSE;
   STATUS[25].EXT.Forced := TRUE;
   STATUS[25].EXT.BIT29 := FALSE;
   STATUS[25].EXT.BIT30 := FALSE;
   STATUS[25].EXT.BIT31 := FALSE;
   STATUS[25].EXT.ModeBit1 := FALSE;
   STATUS[25].EXT.ModeBit2 := FALSE;
   STATUS[25].EXT.ModeBit3 := FALSE;
   STATUS[25].EXT.BIT19 := FALSE;
   STATUS[25].EXT.BIT20 := FALSE;
   STATUS[25].EXT.AlarmSuppressed := FALSE;
   STATUS[25].EXT.AlarmPresent := FALSE;
   STATUS[25].EXT.AlarmFailUnAck := TRUE;
   STATUS[25].Status := 190;
   STATUS[25].TimeStamp := 16#67F1;
   STATUS[26].EXT.AlarmWarnUnAck := FALSE;
   STATUS[26].EXT.AckRequired := FALSE;
   STATUS[26].EXT.Maintanence := FALSE;
   STATUS[26].EXT.Operation := TRUE;
   STATUS[26].EXT.Forced := FALSE;
   STATUS[26].EXT.BIT29 := FALSE;
   STATUS[26].EXT.BIT30 := FALSE;
   STATUS[26].EXT.BIT31 := FALSE;
   STATUS[26].EXT.ModeBit1 := FALSE;
   STATUS[26].EXT.ModeBit2 := FALSE;
   STATUS[26].EXT.ModeBit3 := FALSE;
   STATUS[26].EXT.BIT19 := FALSE;
   STATUS[26].EXT.BIT20 := FALSE;
   STATUS[26].EXT.AlarmSuppressed := TRUE;
   STATUS[26].EXT.AlarmPresent := FALSE;
   STATUS[26].EXT.AlarmFailUnAck := FALSE;
   STATUS[26].Status := 4177;
   STATUS[26].TimeStamp := 16#8D18;
   STATUS[27].EXT.AlarmWarnUnAck := FALSE;
   STATUS[27].EXT.AckRequired := FALSE;
   STATUS[27].EXT.Maintanence := FALSE;
   STATUS[27].EXT.Operation := TRUE;
   STATUS[27].EXT.Forced := FALSE;
   STATUS[27].EXT.BIT29 := FALSE;
   STATUS[27].EXT.BIT30 := FALSE;
   STATUS[27].EXT.BIT31 := FALSE;
   STATUS[27].EXT.ModeBit1 := FALSE;
   STATUS[27].EXT.ModeBit2 := FALSE;
   STATUS[27].EXT.ModeBit3 := FALSE;
   STATUS[27].EXT.BIT19 := FALSE;
   STATUS[27].EXT.BIT20 := FALSE;
   STATUS[27].EXT.AlarmSuppressed := TRUE;
   STATUS[27].EXT.AlarmPresent := FALSE;
   STATUS[27].EXT.AlarmFailUnAck := FALSE;
   STATUS[27].Status := 4177;
   STATUS[27].TimeStamp := 16#873E;
   STATUS[28].EXT.AlarmWarnUnAck := FALSE;
   STATUS[28].EXT.AckRequired := FALSE;
   STATUS[28].EXT.Maintanence := FALSE;
   STATUS[28].EXT.Operation := TRUE;
   STATUS[28].EXT.Forced := FALSE;
   STATUS[28].EXT.BIT29 := FALSE;
   STATUS[28].EXT.BIT30 := FALSE;
   STATUS[28].EXT.BIT31 := FALSE;
   STATUS[28].EXT.ModeBit1 := FALSE;
   STATUS[28].EXT.ModeBit2 := FALSE;
   STATUS[28].EXT.ModeBit3 := FALSE;
   STATUS[28].EXT.BIT19 := FALSE;
   STATUS[28].EXT.BIT20 := FALSE;
   STATUS[28].EXT.AlarmSuppressed := TRUE;
   STATUS[28].EXT.AlarmPresent := FALSE;
   STATUS[28].EXT.AlarmFailUnAck := FALSE;
   STATUS[28].Status := 4177;
   STATUS[28].TimeStamp := 16#8356;
   STATUS[29].EXT.AlarmWarnUnAck := FALSE;
   STATUS[29].EXT.AckRequired := FALSE;
   STATUS[29].EXT.Maintanence := FALSE;
   STATUS[29].EXT.Operation := TRUE;
   STATUS[29].EXT.Forced := FALSE;
   STATUS[29].EXT.BIT29 := FALSE;
   STATUS[29].EXT.BIT30 := FALSE;
   STATUS[29].EXT.BIT31 := FALSE;
   STATUS[29].EXT.ModeBit1 := FALSE;
   STATUS[29].EXT.ModeBit2 := FALSE;
   STATUS[29].EXT.ModeBit3 := FALSE;
   STATUS[29].EXT.BIT19 := FALSE;
   STATUS[29].EXT.BIT20 := FALSE;
   STATUS[29].EXT.AlarmSuppressed := TRUE;
   STATUS[29].EXT.AlarmPresent := FALSE;
   STATUS[29].EXT.AlarmFailUnAck := FALSE;
   STATUS[29].Status := 4177;
   STATUS[29].TimeStamp := 16#8F0F;
   STATUS[30].EXT.AlarmWarnUnAck := FALSE;
   STATUS[30].EXT.AckRequired := FALSE;
   STATUS[30].EXT.Maintanence := FALSE;
   STATUS[30].EXT.Operation := FALSE;
   STATUS[30].EXT.Forced := FALSE;
   STATUS[30].EXT.BIT29 := FALSE;
   STATUS[30].EXT.BIT30 := FALSE;
   STATUS[30].EXT.BIT31 := FALSE;
   STATUS[30].EXT.ModeBit1 := FALSE;
   STATUS[30].EXT.ModeBit2 := FALSE;
   STATUS[30].EXT.ModeBit3 := FALSE;
   STATUS[30].EXT.BIT19 := FALSE;
   STATUS[30].EXT.BIT20 := FALSE;
   STATUS[30].EXT.AlarmSuppressed := TRUE;
   STATUS[30].EXT.AlarmPresent := TRUE;
   STATUS[30].EXT.AlarmFailUnAck := TRUE;
   STATUS[30].Status := 207;
   STATUS[30].TimeStamp := 16#84C0;
   STATUS[31].EXT.AlarmWarnUnAck := FALSE;
   STATUS[31].EXT.AckRequired := FALSE;
   STATUS[31].EXT.Maintanence := FALSE;
   STATUS[31].EXT.Operation := FALSE;
   STATUS[31].EXT.Forced := FALSE;
   STATUS[31].EXT.BIT29 := FALSE;
   STATUS[31].EXT.BIT30 := FALSE;
   STATUS[31].EXT.BIT31 := FALSE;
   STATUS[31].EXT.ModeBit1 := TRUE;
   STATUS[31].EXT.ModeBit2 := TRUE;
   STATUS[31].EXT.ModeBit3 := FALSE;
   STATUS[31].EXT.BIT19 := FALSE;
   STATUS[31].EXT.BIT20 := FALSE;
   STATUS[31].EXT.AlarmSuppressed := FALSE;
   STATUS[31].EXT.AlarmPresent := FALSE;
   STATUS[31].EXT.AlarmFailUnAck := FALSE;
   STATUS[31].Status := 1;
   STATUS[31].TimeStamp := 16#D296;
   STATUS[32].EXT.AlarmWarnUnAck := FALSE;
   STATUS[32].EXT.AckRequired := FALSE;
   STATUS[32].EXT.Maintanence := FALSE;
   STATUS[32].EXT.Operation := FALSE;
   STATUS[32].EXT.Forced := FALSE;
   STATUS[32].EXT.BIT29 := FALSE;
   STATUS[32].EXT.BIT30 := FALSE;
   STATUS[32].EXT.BIT31 := FALSE;
   STATUS[32].EXT.ModeBit1 := FALSE;
   STATUS[32].EXT.ModeBit2 := FALSE;
   STATUS[32].EXT.ModeBit3 := FALSE;
   STATUS[32].EXT.BIT19 := FALSE;
   STATUS[32].EXT.BIT20 := FALSE;
   STATUS[32].EXT.AlarmSuppressed := TRUE;
   STATUS[32].EXT.AlarmPresent := TRUE;
   STATUS[32].EXT.AlarmFailUnAck := TRUE;
   STATUS[32].Status := 201;
   STATUS[32].TimeStamp := 16#3928;
   STATUS[33].EXT.AlarmWarnUnAck := FALSE;
   STATUS[33].EXT.AckRequired := FALSE;
   STATUS[33].EXT.Maintanence := FALSE;
   STATUS[33].EXT.Operation := FALSE;
   STATUS[33].EXT.Forced := TRUE;
   STATUS[33].EXT.BIT29 := FALSE;
   STATUS[33].EXT.BIT30 := FALSE;
   STATUS[33].EXT.BIT31 := FALSE;
   STATUS[33].EXT.ModeBit1 := FALSE;
   STATUS[33].EXT.ModeBit2 := FALSE;
   STATUS[33].EXT.ModeBit3 := FALSE;
   STATUS[33].EXT.BIT19 := FALSE;
   STATUS[33].EXT.BIT20 := FALSE;
   STATUS[33].EXT.AlarmSuppressed := FALSE;
   STATUS[33].EXT.AlarmPresent := FALSE;
   STATUS[33].EXT.AlarmFailUnAck := TRUE;
   STATUS[33].Status := 190;
   STATUS[33].TimeStamp := 16#769D;
   STATUS[34].EXT.AlarmWarnUnAck := FALSE;
   STATUS[34].EXT.AckRequired := FALSE;
   STATUS[34].EXT.Maintanence := FALSE;
   STATUS[34].EXT.Operation := FALSE;
   STATUS[34].EXT.Forced := TRUE;
   STATUS[34].EXT.BIT29 := FALSE;
   STATUS[34].EXT.BIT30 := FALSE;
   STATUS[34].EXT.BIT31 := FALSE;
   STATUS[34].EXT.ModeBit1 := FALSE;
   STATUS[34].EXT.ModeBit2 := FALSE;
   STATUS[34].EXT.ModeBit3 := FALSE;
   STATUS[34].EXT.BIT19 := FALSE;
   STATUS[34].EXT.BIT20 := FALSE;
   STATUS[34].EXT.AlarmSuppressed := FALSE;
   STATUS[34].EXT.AlarmPresent := FALSE;
   STATUS[34].EXT.AlarmFailUnAck := TRUE;
   STATUS[34].Status := 190;
   STATUS[34].TimeStamp := 16#8965;
   STATUS[35].EXT.AlarmWarnUnAck := FALSE;
   STATUS[35].EXT.AckRequired := FALSE;
   STATUS[35].EXT.Maintanence := FALSE;
   STATUS[35].EXT.Operation := FALSE;
   STATUS[35].EXT.Forced := TRUE;
   STATUS[35].EXT.BIT29 := FALSE;
   STATUS[35].EXT.BIT30 := FALSE;
   STATUS[35].EXT.BIT31 := FALSE;
   STATUS[35].EXT.ModeBit1 := FALSE;
   STATUS[35].EXT.ModeBit2 := FALSE;
   STATUS[35].EXT.ModeBit3 := FALSE;
   STATUS[35].EXT.BIT19 := FALSE;
   STATUS[35].EXT.BIT20 := FALSE;
   STATUS[35].EXT.AlarmSuppressed := FALSE;
   STATUS[35].EXT.AlarmPresent := FALSE;
   STATUS[35].EXT.AlarmFailUnAck := TRUE;
   STATUS[35].Status := 190;
   STATUS[35].TimeStamp := 16#1A4E;
   STATUS[36].EXT.AlarmWarnUnAck := FALSE;
   STATUS[36].EXT.AckRequired := FALSE;
   STATUS[36].EXT.Maintanence := FALSE;
   STATUS[36].EXT.Operation := FALSE;
   STATUS[36].EXT.Forced := TRUE;
   STATUS[36].EXT.BIT29 := FALSE;
   STATUS[36].EXT.BIT30 := FALSE;
   STATUS[36].EXT.BIT31 := FALSE;
   STATUS[36].EXT.ModeBit1 := FALSE;
   STATUS[36].EXT.ModeBit2 := FALSE;
   STATUS[36].EXT.ModeBit3 := FALSE;
   STATUS[36].EXT.BIT19 := FALSE;
   STATUS[36].EXT.BIT20 := FALSE;
   STATUS[36].EXT.AlarmSuppressed := FALSE;
   STATUS[36].EXT.AlarmPresent := FALSE;
   STATUS[36].EXT.AlarmFailUnAck := TRUE;
   STATUS[36].Status := 190;
   STATUS[36].TimeStamp := 16#8CD3;
   STATUS[37].EXT.AlarmWarnUnAck := FALSE;
   STATUS[37].EXT.AckRequired := FALSE;
   STATUS[37].EXT.Maintanence := FALSE;
   STATUS[37].EXT.Operation := FALSE;
   STATUS[37].EXT.Forced := TRUE;
   STATUS[37].EXT.BIT29 := FALSE;
   STATUS[37].EXT.BIT30 := FALSE;
   STATUS[37].EXT.BIT31 := FALSE;
   STATUS[37].EXT.ModeBit1 := FALSE;
   STATUS[37].EXT.ModeBit2 := FALSE;
   STATUS[37].EXT.ModeBit3 := FALSE;
   STATUS[37].EXT.BIT19 := FALSE;
   STATUS[37].EXT.BIT20 := FALSE;
   STATUS[37].EXT.AlarmSuppressed := FALSE;
   STATUS[37].EXT.AlarmPresent := FALSE;
   STATUS[37].EXT.AlarmFailUnAck := TRUE;
   STATUS[37].Status := 190;
   STATUS[37].TimeStamp := 16#9023;
   STATUS[38].EXT.AlarmWarnUnAck := FALSE;
   STATUS[38].EXT.AckRequired := FALSE;
   STATUS[38].EXT.Maintanence := FALSE;
   STATUS[38].EXT.Operation := FALSE;
   STATUS[38].EXT.Forced := TRUE;
   STATUS[38].EXT.BIT29 := FALSE;
   STATUS[38].EXT.BIT30 := FALSE;
   STATUS[38].EXT.BIT31 := FALSE;
   STATUS[38].EXT.ModeBit1 := FALSE;
   STATUS[38].EXT.ModeBit2 := FALSE;
   STATUS[38].EXT.ModeBit3 := FALSE;
   STATUS[38].EXT.BIT19 := FALSE;
   STATUS[38].EXT.BIT20 := FALSE;
   STATUS[38].EXT.AlarmSuppressed := FALSE;
   STATUS[38].EXT.AlarmPresent := FALSE;
   STATUS[38].EXT.AlarmFailUnAck := TRUE;
   STATUS[38].Status := 190;
   STATUS[38].TimeStamp := 16#8F9D;
   STATUS[39].EXT.AlarmWarnUnAck := FALSE;
   STATUS[39].EXT.AckRequired := FALSE;
   STATUS[39].EXT.Maintanence := FALSE;
   STATUS[39].EXT.Operation := FALSE;
   STATUS[39].EXT.Forced := TRUE;
   STATUS[39].EXT.BIT29 := FALSE;
   STATUS[39].EXT.BIT30 := FALSE;
   STATUS[39].EXT.BIT31 := FALSE;
   STATUS[39].EXT.ModeBit1 := FALSE;
   STATUS[39].EXT.ModeBit2 := FALSE;
   STATUS[39].EXT.ModeBit3 := FALSE;
   STATUS[39].EXT.BIT19 := FALSE;
   STATUS[39].EXT.BIT20 := FALSE;
   STATUS[39].EXT.AlarmSuppressed := FALSE;
   STATUS[39].EXT.AlarmPresent := FALSE;
   STATUS[39].EXT.AlarmFailUnAck := TRUE;
   STATUS[39].Status := 190;
   STATUS[39].TimeStamp := 16#6CC1;
   STATUS[40].EXT.AlarmWarnUnAck := FALSE;
   STATUS[40].EXT.AckRequired := FALSE;
   STATUS[40].EXT.Maintanence := FALSE;
   STATUS[40].EXT.Operation := FALSE;
   STATUS[40].EXT.Forced := TRUE;
   STATUS[40].EXT.BIT29 := FALSE;
   STATUS[40].EXT.BIT30 := FALSE;
   STATUS[40].EXT.BIT31 := FALSE;
   STATUS[40].EXT.ModeBit1 := FALSE;
   STATUS[40].EXT.ModeBit2 := FALSE;
   STATUS[40].EXT.ModeBit3 := FALSE;
   STATUS[40].EXT.BIT19 := FALSE;
   STATUS[40].EXT.BIT20 := FALSE;
   STATUS[40].EXT.AlarmSuppressed := FALSE;
   STATUS[40].EXT.AlarmPresent := FALSE;
   STATUS[40].EXT.AlarmFailUnAck := TRUE;
   STATUS[40].Status := 190;
   STATUS[40].TimeStamp := 16#77D4;
   STATUS[41].EXT.AlarmWarnUnAck := FALSE;
   STATUS[41].EXT.AckRequired := FALSE;
   STATUS[41].EXT.Maintanence := FALSE;
   STATUS[41].EXT.Operation := FALSE;
   STATUS[41].EXT.Forced := FALSE;
   STATUS[41].EXT.BIT29 := FALSE;
   STATUS[41].EXT.BIT30 := FALSE;
   STATUS[41].EXT.BIT31 := FALSE;
   STATUS[41].EXT.ModeBit1 := FALSE;
   STATUS[41].EXT.ModeBit2 := FALSE;
   STATUS[41].EXT.ModeBit3 := FALSE;
   STATUS[41].EXT.BIT19 := FALSE;
   STATUS[41].EXT.BIT20 := FALSE;
   STATUS[41].EXT.AlarmSuppressed := FALSE;
   STATUS[41].EXT.AlarmPresent := FALSE;
   STATUS[41].EXT.AlarmFailUnAck := FALSE;
   STATUS[41].Status := -22466;
   STATUS[41].TimeStamp := 16#B387;
   STATUS[42].EXT.AlarmWarnUnAck := FALSE;
   STATUS[42].EXT.AckRequired := FALSE;
   STATUS[42].EXT.Maintanence := FALSE;
   STATUS[42].EXT.Operation := FALSE;
   STATUS[42].EXT.Forced := TRUE;
   STATUS[42].EXT.BIT29 := FALSE;
   STATUS[42].EXT.BIT30 := FALSE;
   STATUS[42].EXT.BIT31 := FALSE;
   STATUS[42].EXT.ModeBit1 := FALSE;
   STATUS[42].EXT.ModeBit2 := FALSE;
   STATUS[42].EXT.ModeBit3 := FALSE;
   STATUS[42].EXT.BIT19 := FALSE;
   STATUS[42].EXT.BIT20 := FALSE;
   STATUS[42].EXT.AlarmSuppressed := FALSE;
   STATUS[42].EXT.AlarmPresent := FALSE;
   STATUS[42].EXT.AlarmFailUnAck := TRUE;
   STATUS[42].Status := 190;
   STATUS[42].TimeStamp := 16#9426;
   STATUS[43].EXT.AlarmWarnUnAck := FALSE;
   STATUS[43].EXT.AckRequired := FALSE;
   STATUS[43].EXT.Maintanence := FALSE;
   STATUS[43].EXT.Operation := FALSE;
   STATUS[43].EXT.Forced := TRUE;
   STATUS[43].EXT.BIT29 := FALSE;
   STATUS[43].EXT.BIT30 := FALSE;
   STATUS[43].EXT.BIT31 := FALSE;
   STATUS[43].EXT.ModeBit1 := FALSE;
   STATUS[43].EXT.ModeBit2 := FALSE;
   STATUS[43].EXT.ModeBit3 := FALSE;
   STATUS[43].EXT.BIT19 := FALSE;
   STATUS[43].EXT.BIT20 := FALSE;
   STATUS[43].EXT.AlarmSuppressed := FALSE;
   STATUS[43].EXT.AlarmPresent := FALSE;
   STATUS[43].EXT.AlarmFailUnAck := TRUE;
   STATUS[43].Status := 190;
   STATUS[43].TimeStamp := 16#7177;
   STATUS[44].EXT.AlarmWarnUnAck := FALSE;
   STATUS[44].EXT.AckRequired := FALSE;
   STATUS[44].EXT.Maintanence := FALSE;
   STATUS[44].EXT.Operation := FALSE;
   STATUS[44].EXT.Forced := TRUE;
   STATUS[44].EXT.BIT29 := FALSE;
   STATUS[44].EXT.BIT30 := FALSE;
   STATUS[44].EXT.BIT31 := FALSE;
   STATUS[44].EXT.ModeBit1 := FALSE;
   STATUS[44].EXT.ModeBit2 := FALSE;
   STATUS[44].EXT.ModeBit3 := FALSE;
   STATUS[44].EXT.BIT19 := FALSE;
   STATUS[44].EXT.BIT20 := FALSE;
   STATUS[44].EXT.AlarmSuppressed := FALSE;
   STATUS[44].EXT.AlarmPresent := FALSE;
   STATUS[44].EXT.AlarmFailUnAck := TRUE;
   STATUS[44].Status := 190;
   STATUS[44].TimeStamp := 16#7480;
   STATUS[45].EXT.AlarmWarnUnAck := FALSE;
   STATUS[45].EXT.AckRequired := FALSE;
   STATUS[45].EXT.Maintanence := FALSE;
   STATUS[45].EXT.Operation := FALSE;
   STATUS[45].EXT.Forced := FALSE;
   STATUS[45].EXT.BIT29 := FALSE;
   STATUS[45].EXT.BIT30 := FALSE;
   STATUS[45].EXT.BIT31 := FALSE;
   STATUS[45].EXT.ModeBit1 := FALSE;
   STATUS[45].EXT.ModeBit2 := FALSE;
   STATUS[45].EXT.ModeBit3 := FALSE;
   STATUS[45].EXT.BIT19 := FALSE;
   STATUS[45].EXT.BIT20 := FALSE;
   STATUS[45].EXT.AlarmSuppressed := TRUE;
   STATUS[45].EXT.AlarmPresent := TRUE;
   STATUS[45].EXT.AlarmFailUnAck := TRUE;
   STATUS[45].Status := 201;
   STATUS[45].TimeStamp := 16#3928;
   STATUS[46].EXT.AlarmWarnUnAck := FALSE;
   STATUS[46].EXT.AckRequired := FALSE;
   STATUS[46].EXT.Maintanence := FALSE;
   STATUS[46].EXT.Operation := FALSE;
   STATUS[46].EXT.Forced := TRUE;
   STATUS[46].EXT.BIT29 := FALSE;
   STATUS[46].EXT.BIT30 := FALSE;
   STATUS[46].EXT.BIT31 := FALSE;
   STATUS[46].EXT.ModeBit1 := FALSE;
   STATUS[46].EXT.ModeBit2 := FALSE;
   STATUS[46].EXT.ModeBit3 := FALSE;
   STATUS[46].EXT.BIT19 := FALSE;
   STATUS[46].EXT.BIT20 := FALSE;
   STATUS[46].EXT.AlarmSuppressed := FALSE;
   STATUS[46].EXT.AlarmPresent := FALSE;
   STATUS[46].EXT.AlarmFailUnAck := TRUE;
   STATUS[46].Status := 190;
   STATUS[46].TimeStamp := 16#3D88;
   STATUS[47].EXT.AlarmWarnUnAck := FALSE;
   STATUS[47].EXT.AckRequired := FALSE;
   STATUS[47].EXT.Maintanence := FALSE;
   STATUS[47].EXT.Operation := FALSE;
   STATUS[47].EXT.Forced := TRUE;
   STATUS[47].EXT.BIT29 := FALSE;
   STATUS[47].EXT.BIT30 := FALSE;
   STATUS[47].EXT.BIT31 := FALSE;
   STATUS[47].EXT.ModeBit1 := FALSE;
   STATUS[47].EXT.ModeBit2 := FALSE;
   STATUS[47].EXT.ModeBit3 := FALSE;
   STATUS[47].EXT.BIT19 := FALSE;
   STATUS[47].EXT.BIT20 := FALSE;
   STATUS[47].EXT.AlarmSuppressed := FALSE;
   STATUS[47].EXT.AlarmPresent := FALSE;
   STATUS[47].EXT.AlarmFailUnAck := TRUE;
   STATUS[47].Status := 190;
   STATUS[47].TimeStamp := 16#3AA5;
   STATUS[48].EXT.AlarmWarnUnAck := FALSE;
   STATUS[48].EXT.AckRequired := FALSE;
   STATUS[48].EXT.Maintanence := FALSE;
   STATUS[48].EXT.Operation := FALSE;
   STATUS[48].EXT.Forced := FALSE;
   STATUS[48].EXT.BIT29 := FALSE;
   STATUS[48].EXT.BIT30 := FALSE;
   STATUS[48].EXT.BIT31 := FALSE;
   STATUS[48].EXT.ModeBit1 := FALSE;
   STATUS[48].EXT.ModeBit2 := FALSE;
   STATUS[48].EXT.ModeBit3 := FALSE;
   STATUS[48].EXT.BIT19 := FALSE;
   STATUS[48].EXT.BIT20 := FALSE;
   STATUS[48].EXT.AlarmSuppressed := TRUE;
   STATUS[48].EXT.AlarmPresent := TRUE;
   STATUS[48].EXT.AlarmFailUnAck := TRUE;
   STATUS[48].Status := 201;
   STATUS[48].TimeStamp := 16#3928;
   STATUS[49].EXT.AlarmWarnUnAck := FALSE;
   STATUS[49].EXT.AckRequired := FALSE;
   STATUS[49].EXT.Maintanence := FALSE;
   STATUS[49].EXT.Operation := FALSE;
   STATUS[49].EXT.Forced := TRUE;
   STATUS[49].EXT.BIT29 := FALSE;
   STATUS[49].EXT.BIT30 := FALSE;
   STATUS[49].EXT.BIT31 := FALSE;
   STATUS[49].EXT.ModeBit1 := FALSE;
   STATUS[49].EXT.ModeBit2 := FALSE;
   STATUS[49].EXT.ModeBit3 := FALSE;
   STATUS[49].EXT.BIT19 := FALSE;
   STATUS[49].EXT.BIT20 := FALSE;
   STATUS[49].EXT.AlarmSuppressed := FALSE;
   STATUS[49].EXT.AlarmPresent := FALSE;
   STATUS[49].EXT.AlarmFailUnAck := TRUE;
   STATUS[49].Status := 190;
   STATUS[49].TimeStamp := 16#3CAF;
   STATUS[50].EXT.AlarmWarnUnAck := FALSE;
   STATUS[50].EXT.AckRequired := FALSE;
   STATUS[50].EXT.Maintanence := FALSE;
   STATUS[50].EXT.Operation := FALSE;
   STATUS[50].EXT.Forced := TRUE;
   STATUS[50].EXT.BIT29 := FALSE;
   STATUS[50].EXT.BIT30 := FALSE;
   STATUS[50].EXT.BIT31 := FALSE;
   STATUS[50].EXT.ModeBit1 := FALSE;
   STATUS[50].EXT.ModeBit2 := FALSE;
   STATUS[50].EXT.ModeBit3 := FALSE;
   STATUS[50].EXT.BIT19 := FALSE;
   STATUS[50].EXT.BIT20 := FALSE;
   STATUS[50].EXT.AlarmSuppressed := FALSE;
   STATUS[50].EXT.AlarmPresent := FALSE;
   STATUS[50].EXT.AlarmFailUnAck := TRUE;
   STATUS[50].Status := 190;
   STATUS[50].TimeStamp := 16#3762;
   STATUS[51].EXT.AlarmWarnUnAck := FALSE;
   STATUS[51].EXT.AckRequired := FALSE;
   STATUS[51].EXT.Maintanence := FALSE;
   STATUS[51].EXT.Operation := FALSE;
   STATUS[51].EXT.Forced := TRUE;
   STATUS[51].EXT.BIT29 := FALSE;
   STATUS[51].EXT.BIT30 := FALSE;
   STATUS[51].EXT.BIT31 := FALSE;
   STATUS[51].EXT.ModeBit1 := FALSE;
   STATUS[51].EXT.ModeBit2 := FALSE;
   STATUS[51].EXT.ModeBit3 := FALSE;
   STATUS[51].EXT.BIT19 := FALSE;
   STATUS[51].EXT.BIT20 := FALSE;
   STATUS[51].EXT.AlarmSuppressed := FALSE;
   STATUS[51].EXT.AlarmPresent := FALSE;
   STATUS[51].EXT.AlarmFailUnAck := TRUE;
   STATUS[51].Status := 190;
   STATUS[51].TimeStamp := 16#2B6B;
   STATUS[52].EXT.AlarmWarnUnAck := FALSE;
   STATUS[52].EXT.AckRequired := FALSE;
   STATUS[52].EXT.Maintanence := FALSE;
   STATUS[52].EXT.Operation := FALSE;
   STATUS[52].EXT.Forced := TRUE;
   STATUS[52].EXT.BIT29 := FALSE;
   STATUS[52].EXT.BIT30 := FALSE;
   STATUS[52].EXT.BIT31 := FALSE;
   STATUS[52].EXT.ModeBit1 := FALSE;
   STATUS[52].EXT.ModeBit2 := FALSE;
   STATUS[52].EXT.ModeBit3 := FALSE;
   STATUS[52].EXT.BIT19 := FALSE;
   STATUS[52].EXT.BIT20 := FALSE;
   STATUS[52].EXT.AlarmSuppressed := FALSE;
   STATUS[52].EXT.AlarmPresent := FALSE;
   STATUS[52].EXT.AlarmFailUnAck := TRUE;
   STATUS[52].Status := 190;
   STATUS[52].TimeStamp := 16#2905;
   STATUS[53].EXT.AlarmWarnUnAck := FALSE;
   STATUS[53].EXT.AckRequired := FALSE;
   STATUS[53].EXT.Maintanence := FALSE;
   STATUS[53].EXT.Operation := FALSE;
   STATUS[53].EXT.Forced := TRUE;
   STATUS[53].EXT.BIT29 := FALSE;
   STATUS[53].EXT.BIT30 := FALSE;
   STATUS[53].EXT.BIT31 := FALSE;
   STATUS[53].EXT.ModeBit1 := FALSE;
   STATUS[53].EXT.ModeBit2 := FALSE;
   STATUS[53].EXT.ModeBit3 := FALSE;
   STATUS[53].EXT.BIT19 := FALSE;
   STATUS[53].EXT.BIT20 := FALSE;
   STATUS[53].EXT.AlarmSuppressed := FALSE;
   STATUS[53].EXT.AlarmPresent := FALSE;
   STATUS[53].EXT.AlarmFailUnAck := TRUE;
   STATUS[53].Status := 190;
   STATUS[53].TimeStamp := 16#2ED3;
   STATUS[54].EXT.AlarmWarnUnAck := FALSE;
   STATUS[54].EXT.AckRequired := FALSE;
   STATUS[54].EXT.Maintanence := FALSE;
   STATUS[54].EXT.Operation := FALSE;
   STATUS[54].EXT.Forced := TRUE;
   STATUS[54].EXT.BIT29 := FALSE;
   STATUS[54].EXT.BIT30 := FALSE;
   STATUS[54].EXT.BIT31 := FALSE;
   STATUS[54].EXT.ModeBit1 := FALSE;
   STATUS[54].EXT.ModeBit2 := FALSE;
   STATUS[54].EXT.ModeBit3 := FALSE;
   STATUS[54].EXT.BIT19 := FALSE;
   STATUS[54].EXT.BIT20 := FALSE;
   STATUS[54].EXT.AlarmSuppressed := FALSE;
   STATUS[54].EXT.AlarmPresent := FALSE;
   STATUS[54].EXT.AlarmFailUnAck := TRUE;
   STATUS[54].Status := 190;
   STATUS[54].TimeStamp := 16#326B;
   STATUS[55].EXT.AlarmWarnUnAck := FALSE;
   STATUS[55].EXT.AckRequired := FALSE;
   STATUS[55].EXT.Maintanence := FALSE;
   STATUS[55].EXT.Operation := FALSE;
   STATUS[55].EXT.Forced := TRUE;
   STATUS[55].EXT.BIT29 := FALSE;
   STATUS[55].EXT.BIT30 := FALSE;
   STATUS[55].EXT.BIT31 := FALSE;
   STATUS[55].EXT.ModeBit1 := FALSE;
   STATUS[55].EXT.ModeBit2 := FALSE;
   STATUS[55].EXT.ModeBit3 := FALSE;
   STATUS[55].EXT.BIT19 := FALSE;
   STATUS[55].EXT.BIT20 := FALSE;
   STATUS[55].EXT.AlarmSuppressed := FALSE;
   STATUS[55].EXT.AlarmPresent := FALSE;
   STATUS[55].EXT.AlarmFailUnAck := TRUE;
   STATUS[55].Status := 190;
   STATUS[55].TimeStamp := 16#354C;
   STATUS[56].EXT.AlarmWarnUnAck := FALSE;
   STATUS[56].EXT.AckRequired := FALSE;
   STATUS[56].EXT.Maintanence := FALSE;
   STATUS[56].EXT.Operation := FALSE;
   STATUS[56].EXT.Forced := TRUE;
   STATUS[56].EXT.BIT29 := FALSE;
   STATUS[56].EXT.BIT30 := FALSE;
   STATUS[56].EXT.BIT31 := FALSE;
   STATUS[56].EXT.ModeBit1 := FALSE;
   STATUS[56].EXT.ModeBit2 := FALSE;
   STATUS[56].EXT.ModeBit3 := FALSE;
   STATUS[56].EXT.BIT19 := FALSE;
   STATUS[56].EXT.BIT20 := FALSE;
   STATUS[56].EXT.AlarmSuppressed := FALSE;
   STATUS[56].EXT.AlarmPresent := FALSE;
   STATUS[56].EXT.AlarmFailUnAck := TRUE;
   STATUS[56].Status := 190;
   STATUS[56].TimeStamp := 16#5DA1;
   STATUS[57].EXT.AlarmWarnUnAck := FALSE;
   STATUS[57].EXT.AckRequired := FALSE;
   STATUS[57].EXT.Maintanence := FALSE;
   STATUS[57].EXT.Operation := FALSE;
   STATUS[57].EXT.Forced := TRUE;
   STATUS[57].EXT.BIT29 := FALSE;
   STATUS[57].EXT.BIT30 := FALSE;
   STATUS[57].EXT.BIT31 := FALSE;
   STATUS[57].EXT.ModeBit1 := FALSE;
   STATUS[57].EXT.ModeBit2 := FALSE;
   STATUS[57].EXT.ModeBit3 := FALSE;
   STATUS[57].EXT.BIT19 := FALSE;
   STATUS[57].EXT.BIT20 := FALSE;
   STATUS[57].EXT.AlarmSuppressed := FALSE;
   STATUS[57].EXT.AlarmPresent := FALSE;
   STATUS[57].EXT.AlarmFailUnAck := TRUE;
   STATUS[57].Status := 190;
   STATUS[57].TimeStamp := 16#A396;
   STATUS[58].EXT.AlarmWarnUnAck := FALSE;
   STATUS[58].EXT.AckRequired := FALSE;
   STATUS[58].EXT.Maintanence := FALSE;
   STATUS[58].EXT.Operation := FALSE;
   STATUS[58].EXT.Forced := TRUE;
   STATUS[58].EXT.BIT29 := FALSE;
   STATUS[58].EXT.BIT30 := FALSE;
   STATUS[58].EXT.BIT31 := FALSE;
   STATUS[58].EXT.ModeBit1 := FALSE;
   STATUS[58].EXT.ModeBit2 := FALSE;
   STATUS[58].EXT.ModeBit3 := FALSE;
   STATUS[58].EXT.BIT19 := FALSE;
   STATUS[58].EXT.BIT20 := FALSE;
   STATUS[58].EXT.AlarmSuppressed := FALSE;
   STATUS[58].EXT.AlarmPresent := FALSE;
   STATUS[58].EXT.AlarmFailUnAck := TRUE;
   STATUS[58].Status := 190;
   STATUS[58].TimeStamp := 16#B493;
   STATUS[59].EXT.AlarmWarnUnAck := FALSE;
   STATUS[59].EXT.AckRequired := FALSE;
   STATUS[59].EXT.Maintanence := FALSE;
   STATUS[59].EXT.Operation := FALSE;
   STATUS[59].EXT.Forced := TRUE;
   STATUS[59].EXT.BIT29 := FALSE;
   STATUS[59].EXT.BIT30 := FALSE;
   STATUS[59].EXT.BIT31 := FALSE;
   STATUS[59].EXT.ModeBit1 := FALSE;
   STATUS[59].EXT.ModeBit2 := FALSE;
   STATUS[59].EXT.ModeBit3 := FALSE;
   STATUS[59].EXT.BIT19 := FALSE;
   STATUS[59].EXT.BIT20 := FALSE;
   STATUS[59].EXT.AlarmSuppressed := FALSE;
   STATUS[59].EXT.AlarmPresent := FALSE;
   STATUS[59].EXT.AlarmFailUnAck := TRUE;
   STATUS[59].Status := 190;
   STATUS[59].TimeStamp := 16#E0C9;
   STATUS[60].EXT.AlarmWarnUnAck := FALSE;
   STATUS[60].EXT.AckRequired := FALSE;
   STATUS[60].EXT.Maintanence := FALSE;
   STATUS[60].EXT.Operation := FALSE;
   STATUS[60].EXT.Forced := TRUE;
   STATUS[60].EXT.BIT29 := FALSE;
   STATUS[60].EXT.BIT30 := FALSE;
   STATUS[60].EXT.BIT31 := FALSE;
   STATUS[60].EXT.ModeBit1 := FALSE;
   STATUS[60].EXT.ModeBit2 := FALSE;
   STATUS[60].EXT.ModeBit3 := FALSE;
   STATUS[60].EXT.BIT19 := FALSE;
   STATUS[60].EXT.BIT20 := FALSE;
   STATUS[60].EXT.AlarmSuppressed := FALSE;
   STATUS[60].EXT.AlarmPresent := FALSE;
   STATUS[60].EXT.AlarmFailUnAck := TRUE;
   STATUS[60].Status := 190;
   STATUS[60].TimeStamp := 16#8623;
   STATUS[61].EXT.AlarmWarnUnAck := FALSE;
   STATUS[61].EXT.AckRequired := FALSE;
   STATUS[61].EXT.Maintanence := FALSE;
   STATUS[61].EXT.Operation := FALSE;
   STATUS[61].EXT.Forced := TRUE;
   STATUS[61].EXT.BIT29 := FALSE;
   STATUS[61].EXT.BIT30 := FALSE;
   STATUS[61].EXT.BIT31 := FALSE;
   STATUS[61].EXT.ModeBit1 := FALSE;
   STATUS[61].EXT.ModeBit2 := FALSE;
   STATUS[61].EXT.ModeBit3 := FALSE;
   STATUS[61].EXT.BIT19 := FALSE;
   STATUS[61].EXT.BIT20 := FALSE;
   STATUS[61].EXT.AlarmSuppressed := FALSE;
   STATUS[61].EXT.AlarmPresent := FALSE;
   STATUS[61].EXT.AlarmFailUnAck := TRUE;
   STATUS[61].Status := 190;
   STATUS[61].TimeStamp := 16#8C63;
   STATUS[62].EXT.AlarmWarnUnAck := FALSE;
   STATUS[62].EXT.AckRequired := FALSE;
   STATUS[62].EXT.Maintanence := FALSE;
   STATUS[62].EXT.Operation := FALSE;
   STATUS[62].EXT.Forced := TRUE;
   STATUS[62].EXT.BIT29 := FALSE;
   STATUS[62].EXT.BIT30 := FALSE;
   STATUS[62].EXT.BIT31 := FALSE;
   STATUS[62].EXT.ModeBit1 := FALSE;
   STATUS[62].EXT.ModeBit2 := FALSE;
   STATUS[62].EXT.ModeBit3 := FALSE;
   STATUS[62].EXT.BIT19 := FALSE;
   STATUS[62].EXT.BIT20 := FALSE;
   STATUS[62].EXT.AlarmSuppressed := FALSE;
   STATUS[62].EXT.AlarmPresent := FALSE;
   STATUS[62].EXT.AlarmFailUnAck := TRUE;
   STATUS[62].Status := 190;
   STATUS[62].TimeStamp := 16#894E;
   STATUS[63].EXT.AlarmWarnUnAck := FALSE;
   STATUS[63].EXT.AckRequired := FALSE;
   STATUS[63].EXT.Maintanence := FALSE;
   STATUS[63].EXT.Operation := FALSE;
   STATUS[63].EXT.Forced := TRUE;
   STATUS[63].EXT.BIT29 := FALSE;
   STATUS[63].EXT.BIT30 := FALSE;
   STATUS[63].EXT.BIT31 := FALSE;
   STATUS[63].EXT.ModeBit1 := FALSE;
   STATUS[63].EXT.ModeBit2 := FALSE;
   STATUS[63].EXT.ModeBit3 := FALSE;
   STATUS[63].EXT.BIT19 := FALSE;
   STATUS[63].EXT.BIT20 := FALSE;
   STATUS[63].EXT.AlarmSuppressed := FALSE;
   STATUS[63].EXT.AlarmPresent := FALSE;
   STATUS[63].EXT.AlarmFailUnAck := TRUE;
   STATUS[63].Status := 190;
   STATUS[63].TimeStamp := 16#6CB2;
   STATUS[64].EXT.AlarmWarnUnAck := FALSE;
   STATUS[64].EXT.AckRequired := FALSE;
   STATUS[64].EXT.Maintanence := FALSE;
   STATUS[64].EXT.Operation := FALSE;
   STATUS[64].EXT.Forced := TRUE;
   STATUS[64].EXT.BIT29 := FALSE;
   STATUS[64].EXT.BIT30 := FALSE;
   STATUS[64].EXT.BIT31 := FALSE;
   STATUS[64].EXT.ModeBit1 := FALSE;
   STATUS[64].EXT.ModeBit2 := FALSE;
   STATUS[64].EXT.ModeBit3 := FALSE;
   STATUS[64].EXT.BIT19 := FALSE;
   STATUS[64].EXT.BIT20 := FALSE;
   STATUS[64].EXT.AlarmSuppressed := FALSE;
   STATUS[64].EXT.AlarmPresent := FALSE;
   STATUS[64].EXT.AlarmFailUnAck := TRUE;
   STATUS[64].Status := 190;
   STATUS[64].TimeStamp := 16#7AB9;
   STATUS[65].EXT.AlarmWarnUnAck := FALSE;
   STATUS[65].EXT.AckRequired := FALSE;
   STATUS[65].EXT.Maintanence := FALSE;
   STATUS[65].EXT.Operation := FALSE;
   STATUS[65].EXT.Forced := TRUE;
   STATUS[65].EXT.BIT29 := FALSE;
   STATUS[65].EXT.BIT30 := FALSE;
   STATUS[65].EXT.BIT31 := FALSE;
   STATUS[65].EXT.ModeBit1 := FALSE;
   STATUS[65].EXT.ModeBit2 := FALSE;
   STATUS[65].EXT.ModeBit3 := FALSE;
   STATUS[65].EXT.BIT19 := FALSE;
   STATUS[65].EXT.BIT20 := FALSE;
   STATUS[65].EXT.AlarmSuppressed := FALSE;
   STATUS[65].EXT.AlarmPresent := FALSE;
   STATUS[65].EXT.AlarmFailUnAck := TRUE;
   STATUS[65].Status := 190;
   STATUS[65].TimeStamp := 16#A000;
   STATUS[66].EXT.AlarmWarnUnAck := FALSE;
   STATUS[66].EXT.AckRequired := FALSE;
   STATUS[66].EXT.Maintanence := FALSE;
   STATUS[66].EXT.Operation := FALSE;
   STATUS[66].EXT.Forced := TRUE;
   STATUS[66].EXT.BIT29 := FALSE;
   STATUS[66].EXT.BIT30 := FALSE;
   STATUS[66].EXT.BIT31 := FALSE;
   STATUS[66].EXT.ModeBit1 := FALSE;
   STATUS[66].EXT.ModeBit2 := FALSE;
   STATUS[66].EXT.ModeBit3 := FALSE;
   STATUS[66].EXT.BIT19 := FALSE;
   STATUS[66].EXT.BIT20 := FALSE;
   STATUS[66].EXT.AlarmSuppressed := FALSE;
   STATUS[66].EXT.AlarmPresent := FALSE;
   STATUS[66].EXT.AlarmFailUnAck := TRUE;
   STATUS[66].Status := 190;
   STATUS[66].TimeStamp := 16#ACE3;
   STATUS[67].EXT.AlarmWarnUnAck := FALSE;
   STATUS[67].EXT.AckRequired := FALSE;
   STATUS[67].EXT.Maintanence := FALSE;
   STATUS[67].EXT.Operation := FALSE;
   STATUS[67].EXT.Forced := TRUE;
   STATUS[67].EXT.BIT29 := FALSE;
   STATUS[67].EXT.BIT30 := FALSE;
   STATUS[67].EXT.BIT31 := FALSE;
   STATUS[67].EXT.ModeBit1 := FALSE;
   STATUS[67].EXT.ModeBit2 := FALSE;
   STATUS[67].EXT.ModeBit3 := FALSE;
   STATUS[67].EXT.BIT19 := FALSE;
   STATUS[67].EXT.BIT20 := FALSE;
   STATUS[67].EXT.AlarmSuppressed := FALSE;
   STATUS[67].EXT.AlarmPresent := FALSE;
   STATUS[67].EXT.AlarmFailUnAck := TRUE;
   STATUS[67].Status := 190;
   STATUS[67].TimeStamp := 16#C304;
   STATUS[68].EXT.AlarmWarnUnAck := FALSE;
   STATUS[68].EXT.AckRequired := FALSE;
   STATUS[68].EXT.Maintanence := FALSE;
   STATUS[68].EXT.Operation := FALSE;
   STATUS[68].EXT.Forced := TRUE;
   STATUS[68].EXT.BIT29 := FALSE;
   STATUS[68].EXT.BIT30 := FALSE;
   STATUS[68].EXT.BIT31 := FALSE;
   STATUS[68].EXT.ModeBit1 := FALSE;
   STATUS[68].EXT.ModeBit2 := FALSE;
   STATUS[68].EXT.ModeBit3 := FALSE;
   STATUS[68].EXT.BIT19 := FALSE;
   STATUS[68].EXT.BIT20 := FALSE;
   STATUS[68].EXT.AlarmSuppressed := FALSE;
   STATUS[68].EXT.AlarmPresent := FALSE;
   STATUS[68].EXT.AlarmFailUnAck := TRUE;
   STATUS[68].Status := 190;
   STATUS[68].TimeStamp := 16#7FB7;
   STATUS[69].EXT.AlarmWarnUnAck := FALSE;
   STATUS[69].EXT.AckRequired := FALSE;
   STATUS[69].EXT.Maintanence := FALSE;
   STATUS[69].EXT.Operation := FALSE;
   STATUS[69].EXT.Forced := TRUE;
   STATUS[69].EXT.BIT29 := FALSE;
   STATUS[69].EXT.BIT30 := FALSE;
   STATUS[69].EXT.BIT31 := FALSE;
   STATUS[69].EXT.ModeBit1 := FALSE;
   STATUS[69].EXT.ModeBit2 := FALSE;
   STATUS[69].EXT.ModeBit3 := FALSE;
   STATUS[69].EXT.BIT19 := FALSE;
   STATUS[69].EXT.BIT20 := FALSE;
   STATUS[69].EXT.AlarmSuppressed := FALSE;
   STATUS[69].EXT.AlarmPresent := FALSE;
   STATUS[69].EXT.AlarmFailUnAck := TRUE;
   STATUS[69].Status := 190;
   STATUS[69].TimeStamp := 16#795D;
   STATUS[70].EXT.AlarmWarnUnAck := FALSE;
   STATUS[70].EXT.AckRequired := FALSE;
   STATUS[70].EXT.Maintanence := FALSE;
   STATUS[70].EXT.Operation := FALSE;
   STATUS[70].EXT.Forced := TRUE;
   STATUS[70].EXT.BIT29 := FALSE;
   STATUS[70].EXT.BIT30 := FALSE;
   STATUS[70].EXT.BIT31 := FALSE;
   STATUS[70].EXT.ModeBit1 := FALSE;
   STATUS[70].EXT.ModeBit2 := FALSE;
   STATUS[70].EXT.ModeBit3 := FALSE;
   STATUS[70].EXT.BIT19 := FALSE;
   STATUS[70].EXT.BIT20 := FALSE;
   STATUS[70].EXT.AlarmSuppressed := FALSE;
   STATUS[70].EXT.AlarmPresent := FALSE;
   STATUS[70].EXT.AlarmFailUnAck := TRUE;
   STATUS[70].Status := 190;
   STATUS[70].TimeStamp := 16#7C8E;
   STATUS[71].EXT.AlarmWarnUnAck := FALSE;
   STATUS[71].EXT.AckRequired := FALSE;
   STATUS[71].EXT.Maintanence := FALSE;
   STATUS[71].EXT.Operation := FALSE;
   STATUS[71].EXT.Forced := TRUE;
   STATUS[71].EXT.BIT29 := FALSE;
   STATUS[71].EXT.BIT30 := FALSE;
   STATUS[71].EXT.BIT31 := FALSE;
   STATUS[71].EXT.ModeBit1 := FALSE;
   STATUS[71].EXT.ModeBit2 := FALSE;
   STATUS[71].EXT.ModeBit3 := FALSE;
   STATUS[71].EXT.BIT19 := FALSE;
   STATUS[71].EXT.BIT20 := FALSE;
   STATUS[71].EXT.AlarmSuppressed := FALSE;
   STATUS[71].EXT.AlarmPresent := FALSE;
   STATUS[71].EXT.AlarmFailUnAck := TRUE;
   STATUS[71].Status := 190;
   STATUS[71].TimeStamp := 16#0D7E;
   STATUS[72].EXT.AlarmWarnUnAck := FALSE;
   STATUS[72].EXT.AckRequired := FALSE;
   STATUS[72].EXT.Maintanence := FALSE;
   STATUS[72].EXT.Operation := FALSE;
   STATUS[72].EXT.Forced := TRUE;
   STATUS[72].EXT.BIT29 := FALSE;
   STATUS[72].EXT.BIT30 := FALSE;
   STATUS[72].EXT.BIT31 := FALSE;
   STATUS[72].EXT.ModeBit1 := FALSE;
   STATUS[72].EXT.ModeBit2 := FALSE;
   STATUS[72].EXT.ModeBit3 := FALSE;
   STATUS[72].EXT.BIT19 := FALSE;
   STATUS[72].EXT.BIT20 := FALSE;
   STATUS[72].EXT.AlarmSuppressed := FALSE;
   STATUS[72].EXT.AlarmPresent := FALSE;
   STATUS[72].EXT.AlarmFailUnAck := TRUE;
   STATUS[72].Status := 190;
   STATUS[72].TimeStamp := 16#6FB7;
   STATUS[73].EXT.AlarmWarnUnAck := FALSE;
   STATUS[73].EXT.AckRequired := FALSE;
   STATUS[73].EXT.Maintanence := FALSE;
   STATUS[73].EXT.Operation := FALSE;
   STATUS[73].EXT.Forced := TRUE;
   STATUS[73].EXT.BIT29 := FALSE;
   STATUS[73].EXT.BIT30 := FALSE;
   STATUS[73].EXT.BIT31 := FALSE;
   STATUS[73].EXT.ModeBit1 := FALSE;
   STATUS[73].EXT.ModeBit2 := FALSE;
   STATUS[73].EXT.ModeBit3 := FALSE;
   STATUS[73].EXT.BIT19 := FALSE;
   STATUS[73].EXT.BIT20 := FALSE;
   STATUS[73].EXT.AlarmSuppressed := FALSE;
   STATUS[73].EXT.AlarmPresent := FALSE;
   STATUS[73].EXT.AlarmFailUnAck := TRUE;
   STATUS[73].Status := 190;
   STATUS[73].TimeStamp := 16#7E3F;
   STATUS[74].EXT.AlarmWarnUnAck := FALSE;
   STATUS[74].EXT.AckRequired := FALSE;
   STATUS[74].EXT.Maintanence := FALSE;
   STATUS[74].EXT.Operation := FALSE;
   STATUS[74].EXT.Forced := TRUE;
   STATUS[74].EXT.BIT29 := FALSE;
   STATUS[74].EXT.BIT30 := FALSE;
   STATUS[74].EXT.BIT31 := FALSE;
   STATUS[74].EXT.ModeBit1 := FALSE;
   STATUS[74].EXT.ModeBit2 := FALSE;
   STATUS[74].EXT.ModeBit3 := FALSE;
   STATUS[74].EXT.BIT19 := FALSE;
   STATUS[74].EXT.BIT20 := FALSE;
   STATUS[74].EXT.AlarmSuppressed := FALSE;
   STATUS[74].EXT.AlarmPresent := FALSE;
   STATUS[74].EXT.AlarmFailUnAck := TRUE;
   STATUS[74].Status := 190;
   STATUS[74].TimeStamp := 16#6563;
   STATUS[75].EXT.AlarmWarnUnAck := FALSE;
   STATUS[75].EXT.AckRequired := FALSE;
   STATUS[75].EXT.Maintanence := FALSE;
   STATUS[75].EXT.Operation := FALSE;
   STATUS[75].EXT.Forced := FALSE;
   STATUS[75].EXT.BIT29 := FALSE;
   STATUS[75].EXT.BIT30 := FALSE;
   STATUS[75].EXT.BIT31 := FALSE;
   STATUS[75].EXT.ModeBit1 := FALSE;
   STATUS[75].EXT.ModeBit2 := FALSE;
   STATUS[75].EXT.ModeBit3 := FALSE;
   STATUS[75].EXT.BIT19 := FALSE;
   STATUS[75].EXT.BIT20 := FALSE;
   STATUS[75].EXT.AlarmSuppressed := TRUE;
   STATUS[75].EXT.AlarmPresent := TRUE;
   STATUS[75].EXT.AlarmFailUnAck := TRUE;
   STATUS[75].Status := 214;
   STATUS[75].TimeStamp := 16#3928;
   STATUS[76].EXT.AlarmWarnUnAck := FALSE;
   STATUS[76].EXT.AckRequired := FALSE;
   STATUS[76].EXT.Maintanence := FALSE;
   STATUS[76].EXT.Operation := FALSE;
   STATUS[76].EXT.Forced := FALSE;
   STATUS[76].EXT.BIT29 := FALSE;
   STATUS[76].EXT.BIT30 := FALSE;
   STATUS[76].EXT.BIT31 := FALSE;
   STATUS[76].EXT.ModeBit1 := FALSE;
   STATUS[76].EXT.ModeBit2 := FALSE;
   STATUS[76].EXT.ModeBit3 := FALSE;
   STATUS[76].EXT.BIT19 := FALSE;
   STATUS[76].EXT.BIT20 := FALSE;
   STATUS[76].EXT.AlarmSuppressed := TRUE;
   STATUS[76].EXT.AlarmPresent := TRUE;
   STATUS[76].EXT.AlarmFailUnAck := TRUE;
   STATUS[76].Status := 214;
   STATUS[76].TimeStamp := 16#3928;
   STATUS[77].EXT.AlarmWarnUnAck := FALSE;
   STATUS[77].EXT.AckRequired := FALSE;
   STATUS[77].EXT.Maintanence := FALSE;
   STATUS[77].EXT.Operation := FALSE;
   STATUS[77].EXT.Forced := FALSE;
   STATUS[77].EXT.BIT29 := FALSE;
   STATUS[77].EXT.BIT30 := FALSE;
   STATUS[77].EXT.BIT31 := FALSE;
   STATUS[77].EXT.ModeBit1 := FALSE;
   STATUS[77].EXT.ModeBit2 := FALSE;
   STATUS[77].EXT.ModeBit3 := FALSE;
   STATUS[77].EXT.BIT19 := FALSE;
   STATUS[77].EXT.BIT20 := FALSE;
   STATUS[77].EXT.AlarmSuppressed := TRUE;
   STATUS[77].EXT.AlarmPresent := TRUE;
   STATUS[77].EXT.AlarmFailUnAck := TRUE;
   STATUS[77].Status := 214;
   STATUS[77].TimeStamp := 16#3928;
   STATUS[78].EXT.AlarmWarnUnAck := FALSE;
   STATUS[78].EXT.AckRequired := FALSE;
   STATUS[78].EXT.Maintanence := FALSE;
   STATUS[78].EXT.Operation := FALSE;
   STATUS[78].EXT.Forced := TRUE;
   STATUS[78].EXT.BIT29 := FALSE;
   STATUS[78].EXT.BIT30 := FALSE;
   STATUS[78].EXT.BIT31 := FALSE;
   STATUS[78].EXT.ModeBit1 := FALSE;
   STATUS[78].EXT.ModeBit2 := FALSE;
   STATUS[78].EXT.ModeBit3 := FALSE;
   STATUS[78].EXT.BIT19 := FALSE;
   STATUS[78].EXT.BIT20 := FALSE;
   STATUS[78].EXT.AlarmSuppressed := FALSE;
   STATUS[78].EXT.AlarmPresent := FALSE;
   STATUS[78].EXT.AlarmFailUnAck := TRUE;
   STATUS[78].Status := 190;
   STATUS[78].TimeStamp := 16#72EB;
   STATUS[79].EXT.AlarmWarnUnAck := FALSE;
   STATUS[79].EXT.AckRequired := FALSE;
   STATUS[79].EXT.Maintanence := FALSE;
   STATUS[79].EXT.Operation := FALSE;
   STATUS[79].EXT.Forced := TRUE;
   STATUS[79].EXT.BIT29 := FALSE;
   STATUS[79].EXT.BIT30 := FALSE;
   STATUS[79].EXT.BIT31 := FALSE;
   STATUS[79].EXT.ModeBit1 := FALSE;
   STATUS[79].EXT.ModeBit2 := FALSE;
   STATUS[79].EXT.ModeBit3 := FALSE;
   STATUS[79].EXT.BIT19 := FALSE;
   STATUS[79].EXT.BIT20 := FALSE;
   STATUS[79].EXT.AlarmSuppressed := FALSE;
   STATUS[79].EXT.AlarmPresent := FALSE;
   STATUS[79].EXT.AlarmFailUnAck := TRUE;
   STATUS[79].Status := 190;
   STATUS[79].TimeStamp := 16#6961;
   STATUS[80].EXT.AlarmWarnUnAck := FALSE;
   STATUS[80].EXT.AckRequired := TRUE;
   STATUS[80].EXT.Maintanence := FALSE;
   STATUS[80].EXT.Operation := FALSE;
   STATUS[80].EXT.Forced := FALSE;
   STATUS[80].EXT.BIT29 := FALSE;
   STATUS[80].EXT.BIT30 := FALSE;
   STATUS[80].EXT.BIT31 := FALSE;
   STATUS[80].EXT.ModeBit1 := FALSE;
   STATUS[80].EXT.ModeBit2 := FALSE;
   STATUS[80].EXT.ModeBit3 := FALSE;
   STATUS[80].EXT.BIT19 := FALSE;
   STATUS[80].EXT.BIT20 := FALSE;
   STATUS[80].EXT.AlarmSuppressed := FALSE;
   STATUS[80].EXT.AlarmPresent := FALSE;
   STATUS[80].EXT.AlarmFailUnAck := TRUE;
   STATUS[80].Status := 231;
   STATUS[80].TimeStamp := 16#8854;
   STATUS[81].EXT.AlarmWarnUnAck := FALSE;
   STATUS[81].EXT.AckRequired := FALSE;
   STATUS[81].EXT.Maintanence := FALSE;
   STATUS[81].EXT.Operation := FALSE;
   STATUS[81].EXT.Forced := TRUE;
   STATUS[81].EXT.BIT29 := FALSE;
   STATUS[81].EXT.BIT30 := FALSE;
   STATUS[81].EXT.BIT31 := FALSE;
   STATUS[81].EXT.ModeBit1 := FALSE;
   STATUS[81].EXT.ModeBit2 := FALSE;
   STATUS[81].EXT.ModeBit3 := FALSE;
   STATUS[81].EXT.BIT19 := FALSE;
   STATUS[81].EXT.BIT20 := FALSE;
   STATUS[81].EXT.AlarmSuppressed := FALSE;
   STATUS[81].EXT.AlarmPresent := FALSE;
   STATUS[81].EXT.AlarmFailUnAck := TRUE;
   STATUS[81].Status := 190;
   STATUS[81].TimeStamp := 16#1E88;
   STATUS[82].EXT.AlarmWarnUnAck := FALSE;
   STATUS[82].EXT.AckRequired := FALSE;
   STATUS[82].EXT.Maintanence := FALSE;
   STATUS[82].EXT.Operation := FALSE;
   STATUS[82].EXT.Forced := TRUE;
   STATUS[82].EXT.BIT29 := FALSE;
   STATUS[82].EXT.BIT30 := FALSE;
   STATUS[82].EXT.BIT31 := FALSE;
   STATUS[82].EXT.ModeBit1 := FALSE;
   STATUS[82].EXT.ModeBit2 := FALSE;
   STATUS[82].EXT.ModeBit3 := FALSE;
   STATUS[82].EXT.BIT19 := FALSE;
   STATUS[82].EXT.BIT20 := FALSE;
   STATUS[82].EXT.AlarmSuppressed := FALSE;
   STATUS[82].EXT.AlarmPresent := FALSE;
   STATUS[82].EXT.AlarmFailUnAck := TRUE;
   STATUS[82].Status := 190;
   STATUS[82].TimeStamp := 16#216C;
   STATUS[83].EXT.AlarmWarnUnAck := FALSE;
   STATUS[83].EXT.AckRequired := FALSE;
   STATUS[83].EXT.Maintanence := FALSE;
   STATUS[83].EXT.Operation := FALSE;
   STATUS[83].EXT.Forced := TRUE;
   STATUS[83].EXT.BIT29 := FALSE;
   STATUS[83].EXT.BIT30 := FALSE;
   STATUS[83].EXT.BIT31 := FALSE;
   STATUS[83].EXT.ModeBit1 := FALSE;
   STATUS[83].EXT.ModeBit2 := FALSE;
   STATUS[83].EXT.ModeBit3 := FALSE;
   STATUS[83].EXT.BIT19 := FALSE;
   STATUS[83].EXT.BIT20 := FALSE;
   STATUS[83].EXT.AlarmSuppressed := FALSE;
   STATUS[83].EXT.AlarmPresent := FALSE;
   STATUS[83].EXT.AlarmFailUnAck := TRUE;
   STATUS[83].Status := 190;
   STATUS[83].TimeStamp := 16#2433;
   STATUS[84].EXT.AlarmWarnUnAck := FALSE;
   STATUS[84].EXT.AckRequired := FALSE;
   STATUS[84].EXT.Maintanence := FALSE;
